								
emC_LUC[LUC_Num].SCADA.Out.OperatorMd	:=	emC_LUC[LUC_Num].SM.Out.OperatorMd		;
emC_LUC[LUC_Num].SCADA.Out.AutoMd	:=	emC_LUC[LUC_Num].SM.Out.AutoMd		;
emC_LUC[LUC_Num].SCADA.Out.ManualMd	:=	emC_LUC[LUC_Num].SM.Out.ManualMd		;
emC_LUC[LUC_Num].SCADA.Out.FailedToStartAl	:=	emC_LUC[LUC_Num].SM.Out.FailedToStartAl		;
emC_LUC[LUC_Num].SCADA.Out.FailedToStopAl	:=	emC_LUC[LUC_Num].SM.Out.FailedToStopAl		;
emC_LUC[LUC_Num].SCADA.Out.NonCriticalAl	:=	emC_LUC[LUC_Num].SM.In.NonCriticalAlarm		;
emC_LUC[LUC_Num].SCADA.Out.WarningAl	:=	emC_LUC[LUC_Num].SM.In.Warning		;
emC_LUC[LUC_Num].SCADA.Out.CriticalAl	:=	emC_LUC[LUC_Num].SM.In.CriticalAlarm		;
emC_LUC[LUC_Num].SCADA.Out.HealthySt	:=	emC_LUC[LUC_Num].SM.In.HealthySt		;
emC_LUC[LUC_Num].SCADA.Out.OnlineSt	:=	emC_LUC[LUC_Num].SM.In.OnlineSt		;
emC_LUC[LUC_Num].SCADA.Out.RunningSt	:=	emC_LUC[LUC_Num].SM.In.RunningSt		;
emC_LUC[LUC_Num].SCADA.Out.BatEmergencyStop	:=	emC_LUC[LUC_Num].BattPLC.CtrlLo.Out.Batt_Sys.Alarm.EStopAl     		;
emC_LUC[LUC_Num].SCADA.Out.BatInitializeSt	:=	emC_LUC[LUC_Num].BattPLC.CtrlLo.Out.Batt_Sys.BattSMState.BatInitializeSt		;
emC_LUC[LUC_Num].SCADA.Out.BatNotReadySt	:=	emC_LUC[LUC_Num].BattPLC.CtrlLo.Out.Batt_Sys.BattSMState.BatNotReadySt		;
emC_LUC[LUC_Num].SCADA.Out.BatReadySt	:=	emC_LUC[LUC_Num].BattPLC.CtrlLo.Out.Batt_Sys.BattSMState.BatReadySt		;
emC_LUC[LUC_Num].SCADA.Out.BatStartingSt	:=	emC_LUC[LUC_Num].BattPLC.CtrlLo.Out.Batt_Sys.BattSMState.BatStartingSt		;
emC_LUC[LUC_Num].SCADA.Out.BatOnlineSt	:=	emC_LUC[LUC_Num].BattPLC.CtrlLo.Out.Batt_Sys.BattSMState.BatOnlineSt		;
emC_LUC[LUC_Num].SCADA.Out.BatStoppingSt	:=	emC_LUC[LUC_Num].BattPLC.CtrlLo.Out.Batt_Sys.BattSMState.BatStoppingSt		;
emC_LUC[LUC_Num].SCADA.Out.BmsChargingSt	:=	emC_LUC[LUC_Num].BattPLC.CtrlLo.Out.Batt_Sys.BMS_Mode.ChargingSt     		;
emC_LUC[LUC_Num].SCADA.Out.BmsDischargingSt	:=	emC_LUC[LUC_Num].BattPLC.CtrlLo.Out.Batt_Sys.BMS_Mode.DischargingSt     		;
emC_LUC[LUC_Num].SCADA.Out.BattRunningSt	:=	emC_LUC[LUC_Num].BattPLC.CtrlLo.Out.Batt_Sys.BMS_Mode.BattRunningSt     		;
emC_LUC[LUC_Num].SCADA.Out.BmsRkPartOnlineSt	:=	emC_LUC[LUC_Num].BattPLC.CtrlLo.Out.Batt_Sys.BMS_Mode.RkPartOnlineSt     		;
emC_LUC[LUC_Num].SCADA.Out.BmsEStopSPDSt	:=	emC_LUC[LUC_Num].BattPLC.CtrlLo.Out.Batt_Sys.BMS_Mode.EStopSPDSt     		;
emC_LUC[LUC_Num].SCADA.Out.BmsEStopProtSt	:=	emC_LUC[LUC_Num].BattPLC.CtrlLo.Out.Batt_Sys.BMS_Mode.EStopProtSt     		;
emC_LUC[LUC_Num].SCADA.Out.BmsEStopPartSt	:=	emC_LUC[LUC_Num].BattPLC.CtrlLo.Out.Batt_Sys.BMS_Mode.EStopPartSt     		;
emC_LUC[LUC_Num].SCADA.Out.BmsHealthySt	:=	emC_LUC[LUC_Num].BattPLC.CtrlLo.Out.Batt_Sys.Alarm.HealthySt     		;
emC_LUC[LUC_Num].SCADA.Out.BmsFireSysOkSt	:=	emC_LUC[LUC_Num].BattPLC.CtrlLo.Out.Batt_Sys.Alarm.FireSysOkSt     		;
emC_LUC[LUC_Num].SCADA.Out.BmsCriticalAl	:=	emC_LUC[LUC_Num].BattPLC.CtrlLo.Out.Batt_Sys.Alarm.CriticalAl		;
emC_LUC[LUC_Num].SCADA.Out.BmsNonCriticalAl	:=	emC_LUC[LUC_Num].BattPLC.CtrlLo.Out.Batt_Sys.Alarm.NonCriticalAl		;
emC_LUC[LUC_Num].SCADA.Out.BmsWarningAl	:=	emC_LUC[LUC_Num].BattPLC.CtrlLo.Out.Batt_Sys.Alarm.WarningAl		;
emC_LUC[LUC_Num].SCADA.Out.BmsStateTOUT	:=	emC_LUC[LUC_Num].BattPLC.CtrlLo.Out.Batt_Sys.Alarm.StateTOUT		;
emC_LUC[LUC_Num].SCADA.Out.BmsInitCommsFail	:=	emC_LUC[LUC_Num].BattPLC.CtrlLo.Out.Batt_Sys.Alarm.InitCommsFail		;
emC_LUC[LUC_Num].SCADA.Out.BmsMinRkCloseFail	:=	emC_LUC[LUC_Num].BattPLC.CtrlLo.Out.Batt_Sys.Alarm.MinRkCloseFail		;
emC_LUC[LUC_Num].SCADA.Out.BmsRkTripStart	:=	emC_LUC[LUC_Num].BattPLC.CtrlLo.Out.Batt_Sys.Alarm.RkTripStart		;
emC_LUC[LUC_Num].SCADA.Out.BmsMinRkOnlineFail	:=	emC_LUC[LUC_Num].BattPLC.CtrlLo.Out.Batt_Sys.Alarm.MinRkOnlineFail		;
emC_LUC[LUC_Num].SCADA.Out.BmsRkFailToOpen	:=	emC_LUC[LUC_Num].BattPLC.CtrlLo.Out.Batt_Sys.Alarm.RkFailToOpen		;
emC_LUC[LUC_Num].SCADA.Out.BmsSysFireAl	:=	emC_LUC[LUC_Num].BattPLC.CtrlLo.Out.Batt_Sys.Alarm.SysFireAl		;
emC_LUC[LUC_Num].SCADA.Out.BmsBmsLostCommsAl	:=	emC_LUC[LUC_Num].BattPLC.CtrlLo.Out.Batt_Sys.Alarm.BmsLostCommsAl		;
emC_LUC[LUC_Num].SCADA.Out.BmsBankFault	:=	emC_LUC[LUC_Num].BattPLC.CtrlLo.Out.Batt_Sys.Alarm.BankFault		;
emC_LUC[LUC_Num].SCADA.Out.BmsEStopAl	:=	emC_LUC[LUC_Num].BattPLC.CtrlLo.Out.Batt_Sys.Alarm.EStopAl		;
emC_LUC[LUC_Num].SCADA.Out.BmsExtReadyStNotSetAl	:=	emC_LUC[LUC_Num].BattPLC.CtrlLo.Out.Batt_Sys.Alarm.ExtReadyStNotSetAl		;
emC_LUC[LUC_Num].SCADA.Out.BattUSyncErrAl	:=	emC_LUC[LUC_Num].BattPLC.CtrlLo.Out.Batt_Sys.Alarm.BattUSyncErrAl		;
emC_LUC[LUC_Num].SCADA.Out.BmsRkFail2Cls	:=	emC_LUC[LUC_Num].BattPLC.CtrlLo.Out.Batt_Sys.Alarm.RkFail2Cls		;
emC_LUC[LUC_Num].SCADA.Out.BmsRkCntrFailAl	:=	emC_LUC[LUC_Num].BattPLC.CtrlLo.Out.Batt_Sys.Alarm.RkCntrFailAl		;
emC_LUC[LUC_Num].SCADA.Out.BmsRTUComAl	:=	emC_LUC[LUC_Num].BattPLC.CtrlLo.Out.Batt_Sys.BMSAlarmSummary.RTUComAl		;
emC_LUC[LUC_Num].SCADA.Out.BmsRTUComFlt	:=	emC_LUC[LUC_Num].BattPLC.CtrlLo.Out.Batt_Sys.BMSAlarmSummary.RTUComFlt		;
emC_LUC[LUC_Num].SCADA.Out.BmsRkVoltImbAl	:=	emC_LUC[LUC_Num].BattPLC.CtrlLo.Out.Batt_Sys.BMSAlarmSummary.RkVoltImbAl		;
emC_LUC[LUC_Num].SCADA.Out.BmsSysStopAl	:=	emC_LUC[LUC_Num].BattPLC.CtrlLo.Out.Batt_Sys.BMSAlarmSummary.SysStopAl		;
emC_LUC[LUC_Num].SCADA.Out.BmsModuleUnderTempAl	:=	emC_LUC[LUC_Num].BattPLC.CtrlLo.Out.Batt_Sys.BMSAlarm.ModuleUnderTempAl		;
emC_LUC[LUC_Num].SCADA.Out.BmsModuleOverTempAl	:=	emC_LUC[LUC_Num].BattPLC.CtrlLo.Out.Batt_Sys.BMSAlarm.ModuleOverTempAl		;
emC_LUC[LUC_Num].SCADA.Out.BmsModuleUnVoltAl	:=	emC_LUC[LUC_Num].BattPLC.CtrlLo.Out.Batt_Sys.BMSAlarm.ModuleUnVoltAl		;
emC_LUC[LUC_Num].SCADA.Out.BmsModuleOvVoltAl	:=	emC_LUC[LUC_Num].BattPLC.CtrlLo.Out.Batt_Sys.BMSAlarm.ModuleOvVoltAl		;
emC_LUC[LUC_Num].SCADA.Out.BmsRackVoltRegAl	:=	emC_LUC[LUC_Num].BattPLC.CtrlLo.Out.Batt_Sys.BMSAlarm.RackVoltRegAl		;
emC_LUC[LUC_Num].SCADA.Out.BmsRackTempRegAl	:=	emC_LUC[LUC_Num].BattPLC.CtrlLo.Out.Batt_Sys.BMSAlarm.RackTempRegAl		;
emC_LUC[LUC_Num].SCADA.Out.BmsAuxProtAl	:=	emC_LUC[LUC_Num].BattPLC.CtrlLo.Out.Batt_Sys.BMSAlarm.AuxProtAl		;
emC_LUC[LUC_Num].SCADA.Out.BmsChargeOperLimAl	:=	emC_LUC[LUC_Num].BattPLC.CtrlLo.Out.Batt_Sys.BMSAlarm.ChargeOperLimAl		;
emC_LUC[LUC_Num].SCADA.Out.BmsDischargeOperLimAl	:=	emC_LUC[LUC_Num].BattPLC.CtrlLo.Out.Batt_Sys.BMSAlarm.DischargeOperLimAl		;
emC_LUC[LUC_Num].SCADA.Out.BmsRackUnVoltAl	:=	emC_LUC[LUC_Num].BattPLC.CtrlLo.Out.Batt_Sys.BMSAlarm.RackUnVoltAl		;
emC_LUC[LUC_Num].SCADA.Out.BmsRackOvVoltAl	:=	emC_LUC[LUC_Num].BattPLC.CtrlLo.Out.Batt_Sys.BMSAlarm.RackOvVoltAl		;
emC_LUC[LUC_Num].SCADA.Out.BmsRackCommsAl	:=	emC_LUC[LUC_Num].BattPLC.CtrlLo.Out.Batt_Sys.BMSAlarm.RackCommsAl		;
emC_LUC[LUC_Num].SCADA.Out.BmsTrayCommsAl	:=	emC_LUC[LUC_Num].BattPLC.CtrlLo.Out.Batt_Sys.BMSAlarm.TrayCommsAl		;
emC_LUC[LUC_Num].SCADA.Out.BmsDcCntrSensor1Al	:=	emC_LUC[LUC_Num].BattPLC.CtrlLo.Out.Batt_Sys.BMSAlarm.DcCntrSensor1Al		;
emC_LUC[LUC_Num].SCADA.Out.BmsDcCntrSensor2Al	:=	emC_LUC[LUC_Num].BattPLC.CtrlLo.Out.Batt_Sys.BMSAlarm.DcCntrSensor2Al		;
emC_LUC[LUC_Num].SCADA.Out.BmsFanFailAl	:=	emC_LUC[LUC_Num].BattPLC.CtrlLo.Out.Batt_Sys.BMSAlarm.FanFailAl		;
emC_LUC[LUC_Num].SCADA.Out.BmsChargeOverCurrentAl	:=	emC_LUC[LUC_Num].BattPLC.CtrlLo.Out.Batt_Sys.BMSAlarm.ChargeOverCurrentAl		;
emC_LUC[LUC_Num].SCADA.Out.BmsDisChargeOverCurrentAl	:=	emC_LUC[LUC_Num].BattPLC.CtrlLo.Out.Batt_Sys.BMSAlarm.DisChargeOverCurrentAl		;
emC_LUC[LUC_Num].SCADA.Out.BmsRackVSenseDiffAl	:=	emC_LUC[LUC_Num].BattPLC.CtrlLo.Out.Batt_Sys.BMSAlarm.RackVSenseDiffAl		;
emC_LUC[LUC_Num].SCADA.Out.BmsRackFuseFailAl	:=	emC_LUC[LUC_Num].BattPLC.CtrlLo.Out.Batt_Sys.BMSAlarm.RackFuseFailAl		;
emC_LUC[LUC_Num].SCADA.Out.BmsRackCurrentSenserFailAl	:=	emC_LUC[LUC_Num].BattPLC.CtrlLo.Out.Batt_Sys.BMSAlarm.RackCurrentSenserFailAl		;
emC_LUC[LUC_Num].SCADA.Out.BmsRackPermanentUVAl	:=	emC_LUC[LUC_Num].BattPLC.CtrlLo.Out.Batt_Sys.BMSAlarm.RackPermanentUVAl		;
emC_LUC[LUC_Num].SCADA.Out.BmsDcCntr1Al	:=	emC_LUC[LUC_Num].BattPLC.CtrlLo.Out.Batt_Sys.BMSAlarm.DcCntr1Al		;
emC_LUC[LUC_Num].SCADA.Out.BmsDcCntr2Al	:=	emC_LUC[LUC_Num].BattPLC.CtrlLo.Out.Batt_Sys.BMSAlarm.DcCntr2Al		;
emC_LUC[LUC_Num].SCADA.Out.BmsDcSwCntFailAl	:=	emC_LUC[LUC_Num].BattPLC.CtrlLo.Out.Batt_Sys.BMSAlarm.DcSwCntFailAl		;
emC_LUC[LUC_Num].SCADA.Out.BmsCellVoltSenFailAl	:=	emC_LUC[LUC_Num].BattPLC.CtrlLo.Out.Batt_Sys.BMSAlarm.CellVoltSenFailAl		;
emC_LUC[LUC_Num].SCADA.Out.BmsDCFuseSenserFailAl	:=	emC_LUC[LUC_Num].BattPLC.CtrlLo.Out.Batt_Sys.BMSAlarm.DCFuseSenserFailAl		;
emC_LUC[LUC_Num].SCADA.Out.BmsModuleUnderTempProt	:=	emC_LUC[LUC_Num].BattPLC.CtrlLo.Out.Batt_Sys.BMSProt.ModuleUnderTempAl		;
emC_LUC[LUC_Num].SCADA.Out.BmsModuleOverTempProt	:=	emC_LUC[LUC_Num].BattPLC.CtrlLo.Out.Batt_Sys.BMSProt.ModuleOverTempAl		;
emC_LUC[LUC_Num].SCADA.Out.BmsModuleUnVoltProt	:=	emC_LUC[LUC_Num].BattPLC.CtrlLo.Out.Batt_Sys.BMSProt.ModuleUnVoltAl		;
emC_LUC[LUC_Num].SCADA.Out.BmsModuleOvVoltProt	:=	emC_LUC[LUC_Num].BattPLC.CtrlLo.Out.Batt_Sys.BMSProt.ModuleOvVoltAl		;
emC_LUC[LUC_Num].SCADA.Out.BmsRackVoltRegProt	:=	emC_LUC[LUC_Num].BattPLC.CtrlLo.Out.Batt_Sys.BMSProt.RackVoltRegAl		;
emC_LUC[LUC_Num].SCADA.Out.BmsRackTempRegProt	:=	emC_LUC[LUC_Num].BattPLC.CtrlLo.Out.Batt_Sys.BMSProt.RackTempRegAl		;
emC_LUC[LUC_Num].SCADA.Out.BmsAuxProtProt	:=	emC_LUC[LUC_Num].BattPLC.CtrlLo.Out.Batt_Sys.BMSProt.AuxProtAl		;
emC_LUC[LUC_Num].SCADA.Out.BmsChargeOperLimProt	:=	emC_LUC[LUC_Num].BattPLC.CtrlLo.Out.Batt_Sys.BMSProt.ChargeOperLimAl		;
emC_LUC[LUC_Num].SCADA.Out.BmsDischargeOperLimProt	:=	emC_LUC[LUC_Num].BattPLC.CtrlLo.Out.Batt_Sys.BMSProt.DischargeOperLimAl		;
emC_LUC[LUC_Num].SCADA.Out.BmsRackUnVoltProt	:=	emC_LUC[LUC_Num].BattPLC.CtrlLo.Out.Batt_Sys.BMSProt.RackUnVoltAl		;
emC_LUC[LUC_Num].SCADA.Out.BmsRackOvVoltProt	:=	emC_LUC[LUC_Num].BattPLC.CtrlLo.Out.Batt_Sys.BMSProt.RackOvVoltAl		;
emC_LUC[LUC_Num].SCADA.Out.BmsRackCommsProt	:=	emC_LUC[LUC_Num].BattPLC.CtrlLo.Out.Batt_Sys.BMSProt.RackCommsAl		;
emC_LUC[LUC_Num].SCADA.Out.BmsTrayCommsProt	:=	emC_LUC[LUC_Num].BattPLC.CtrlLo.Out.Batt_Sys.BMSProt.TrayCommsAl		;
emC_LUC[LUC_Num].SCADA.Out.BmsDcCntrSensor1Prot	:=	emC_LUC[LUC_Num].BattPLC.CtrlLo.Out.Batt_Sys.BMSProt.DcCntrSensor1Al		;
emC_LUC[LUC_Num].SCADA.Out.BmsDcCntrSensor2Prot	:=	emC_LUC[LUC_Num].BattPLC.CtrlLo.Out.Batt_Sys.BMSProt.DcCntrSensor2Al		;
emC_LUC[LUC_Num].SCADA.Out.BmsFanFailProt	:=	emC_LUC[LUC_Num].BattPLC.CtrlLo.Out.Batt_Sys.BMSProt.FanFailAl		;
emC_LUC[LUC_Num].SCADA.Out.BmsChargeOverCurrentProt	:=	emC_LUC[LUC_Num].BattPLC.CtrlLo.Out.Batt_Sys.BMSProt.ChargeOverCurrentAl		;
emC_LUC[LUC_Num].SCADA.Out.BmsDisChargeOverCurrentProt	:=	emC_LUC[LUC_Num].BattPLC.CtrlLo.Out.Batt_Sys.BMSProt.DisChargeOverCurrentAl		;
emC_LUC[LUC_Num].SCADA.Out.BmsRackVSenseDiffProt	:=	emC_LUC[LUC_Num].BattPLC.CtrlLo.Out.Batt_Sys.BMSProt.RackVSenseDiffAl		;
emC_LUC[LUC_Num].SCADA.Out.BmsRackFuseFailProt	:=	emC_LUC[LUC_Num].BattPLC.CtrlLo.Out.Batt_Sys.BMSProt.RackFuseFailAl		;
emC_LUC[LUC_Num].SCADA.Out.BmsRackCurrentSenserFailProt	:=	emC_LUC[LUC_Num].BattPLC.CtrlLo.Out.Batt_Sys.BMSProt.RackCurrentSenserFailAl		;
emC_LUC[LUC_Num].SCADA.Out.BmsRackPermanentUVProt	:=	emC_LUC[LUC_Num].BattPLC.CtrlLo.Out.Batt_Sys.BMSProt.RackPermanentUVAl		;
emC_LUC[LUC_Num].SCADA.Out.BmsDcCntr1Prot	:=	emC_LUC[LUC_Num].BattPLC.CtrlLo.Out.Batt_Sys.BMSProt.DcCntr1Al		;
emC_LUC[LUC_Num].SCADA.Out.BmsDcCntr2Prot	:=	emC_LUC[LUC_Num].BattPLC.CtrlLo.Out.Batt_Sys.BMSProt.DcCntr2Al		;
emC_LUC[LUC_Num].SCADA.Out.BmsDcSwCntFailProt	:=	emC_LUC[LUC_Num].BattPLC.CtrlLo.Out.Batt_Sys.BMSProt.DcSwCntFailAl		;
emC_LUC[LUC_Num].SCADA.Out.BmsCellVoltSenFailProt	:=	emC_LUC[LUC_Num].BattPLC.CtrlLo.Out.Batt_Sys.BMSProt.CellVoltSenFailAl		;
emC_LUC[LUC_Num].SCADA.Out.BmsDCFuseSenserFailProt	:=	emC_LUC[LUC_Num].BattPLC.CtrlLo.Out.Batt_Sys.BMSProt.DCFuseSenserFailAl		;
								
for i:=1 to emC_LUC[LUC_Num].BattPLC.Pa.NbOfRackPa	DO	
	emC_LUC[LUC_Num].SCADA.Out.Rk[i].OnlineSt	:=	emC_LUC[LUC_Num].BattPLC.CtrlLo.Out.Batt_Rack.Batt_Rack_Array[i].Status.RkOnlineSt	;
	emC_LUC[LUC_Num].SCADA.Out.Rk[i].OnlineSt	:=	emC_LUC[LUC_Num].BattPLC.CtrlLo.Out.Batt_Rack.Batt_Rack_Array[i].Status.RkOnlineSt	;
	emC_LUC[LUC_Num].SCADA.Out.Rk[i].FaultSt	:=	emC_LUC[LUC_Num].BattPLC.CtrlLo.Out.Batt_Rack.Batt_Rack_Array[i].Alarm.RkCriticalAl OR emC_LUC[LUC_Num].BattPLC.CtrlLo.Out.Batt_Rack.Batt_Rack_Array[i].Alarm.RkNonCriticalAl ;
	emC_LUC[LUC_Num].SCADA.Out.Rk[i].SoCAct	:=	emC_LUC[LUC_Num].BattPLC.CtrlLo.Out.Batt_Rack.Batt_Rack_Array[i].Measure.SoCAct	;
	emC_LUC[LUC_Num].SCADA.Out.Rk[i].SoHAct	:=	emC_LUC[LUC_Num].BattPLC.CtrlLo.Out.Batt_Rack.Batt_Rack_Array[i].Measure.SoHAct	;
	emC_LUC[LUC_Num].SCADA.Out.Rk[i].UAct	:=	emC_LUC[LUC_Num].BattPLC.CtrlLo.Out.Batt_Rack.Batt_Rack_Array[i].Measure.UAct	;
	emC_LUC[LUC_Num].SCADA.Out.Rk[i].IAct	:=	emC_LUC[LUC_Num].BattPLC.CtrlLo.Out.Batt_Rack.Batt_Rack_Array[i].Measure.IAct	;
	emC_LUC[LUC_Num].SCADA.Out.Rk[i].TempAct	:=	emC_LUC[LUC_Num].BattPLC.CtrlLo.Out.Batt_Rack.Batt_Rack_Array[i].Measure.CellAvgTAct	;
END_FOR;
								
emC_LUC[LUC_Num].SCADA.Out.GCRunningSt	:=	emC_LUC[LUC_Num].emPs.PS.GCRunningSt		;
emC_LUC[LUC_Num].SCADA.Out.GCHealthy	:=	emC_LUC[LUC_Num].emPs.PS.GCHealthy		;
emC_LUC[LUC_Num].SCADA.Out.GCStartingSt	:=	emC_LUC[LUC_Num].emPs.PS.GCStartingSt		;
emC_LUC[LUC_Num].SCADA.Out.GCReadySt	:=	emC_LUC[LUC_Num].emPs.PS.GCReadySt		;
emC_LUC[LUC_Num].SCADA.Out.GCGridFollowing	:=	emC_LUC[LUC_Num].emPs.PS.GCGridFollowing		;
emC_LUC[LUC_Num].SCADA.Out.GCFaultSt	:=	emC_LUC[LUC_Num].emPs.PS.GCFaultSt		;
emC_LUC[LUC_Num].SCADA.Out.GCGridForming	:=	emC_LUC[LUC_Num].emPs.PS.GCGridForming		;
emC_LUC[LUC_Num].SCADA.Out.GCAreaEPSLost	:=	emC_LUC[LUC_Num].emPs.PS.GCAreaEPSLost		;
emC_LUC[LUC_Num].SCADA.Out.GCChargingSt	:=	emC_LUC[LUC_Num].emPs.PS.GCChargingSt		;
emC_LUC[LUC_Num].SCADA.Out.GCRideThru	:=	emC_LUC[LUC_Num].emPs.PS.GCRideThru		;
emC_LUC[LUC_Num].SCADA.Out.GCTransitionActiveSt	:=	emC_LUC[LUC_Num].emPs.PS.GCTransitionActiveSt		;
emC_LUC[LUC_Num].SCADA.Out.GCGndFault	:=	emC_LUC[LUC_Num].emPs.PS.GCGndFault		;
emC_LUC[LUC_Num].SCADA.Out.GCDCOverU	:=	emC_LUC[LUC_Num].emPs.PS.GCDCOverU		;
emC_LUC[LUC_Num].SCADA.Out.GCACDisconnect	:=	emC_LUC[LUC_Num].emPs.PS.GCACDisconnect		;
emC_LUC[LUC_Num].SCADA.Out.GCDCDisconnect	:=	emC_LUC[LUC_Num].emPs.PS.GCDCDisconnect		;
emC_LUC[LUC_Num].SCADA.Out.GCDCGridDisconnect	:=	emC_LUC[LUC_Num].emPs.PS.GCDCGridDisconnect		;
emC_LUC[LUC_Num].SCADA.Out.GCCabinetOpen	:=	emC_LUC[LUC_Num].emPs.PS.GCCabinetOpen		;
emC_LUC[LUC_Num].SCADA.Out.GCManualShutdown	:=	emC_LUC[LUC_Num].emPs.PS.GCManualShutdown		;
emC_LUC[LUC_Num].SCADA.Out.GCOverTemp	:=	emC_LUC[LUC_Num].emPs.PS.GCOverTemp		;
emC_LUC[LUC_Num].SCADA.Out.GCOverF	:=	emC_LUC[LUC_Num].emPs.PS.GCOverF		;
emC_LUC[LUC_Num].SCADA.Out.GCUnderF	:=	emC_LUC[LUC_Num].emPs.PS.GCUnderF		;
emC_LUC[LUC_Num].SCADA.Out.GCACOverVolt	:=	emC_LUC[LUC_Num].emPs.PS.GCACOverVolt		;
emC_LUC[LUC_Num].SCADA.Out.GCACUnderVolt	:=	emC_LUC[LUC_Num].emPs.PS.GCACUnderVolt		;
emC_LUC[LUC_Num].SCADA.Out.GCBlownFuse	:=	emC_LUC[LUC_Num].emPs.PS.GCBlownFuse		;
emC_LUC[LUC_Num].SCADA.Out.GCUnderTemp	:=	emC_LUC[LUC_Num].emPs.PS.GCUnderTemp		;
emC_LUC[LUC_Num].SCADA.Out.GCMemLoss	:=	emC_LUC[LUC_Num].emPs.PS.GCMemLoss		;
emC_LUC[LUC_Num].SCADA.Out.GCHWTestFailed	:=	emC_LUC[LUC_Num].emPs.PS.GCHWTestFailed		;
emC_LUC[LUC_Num].SCADA.Out.GCABBCtrlWrongConfig	:=	emC_LUC[LUC_Num].emPs.PS.GCABBCtrlWrongConfig		;
emC_LUC[LUC_Num].SCADA.Out.GCABBCtrlReady	:=	emC_LUC[LUC_Num].emPs.PS.GCABBCtrlReady		;
emC_LUC[LUC_Num].SCADA.Out.GCABBCtrlStartingSt	:=	emC_LUC[LUC_Num].emPs.PS.GCABBCtrlStartingSt		;
emC_LUC[LUC_Num].SCADA.Out.GCABBCtrlVGMActiveSt	:=	emC_LUC[LUC_Num].emPs.PS.GCABBCtrlVGMActiveSt		;
emC_LUC[LUC_Num].SCADA.Out.GCABBCtrlGSMActiveSt	:=	emC_LUC[LUC_Num].emPs.PS.GCABBCtrlGSMActiveSt		;
emC_LUC[LUC_Num].SCADA.Out.GCABBCtrlError	:=	emC_LUC[LUC_Num].emPs.PS.GCABBCtrlError		;
emC_LUC[LUC_Num].SCADA.Out.GCABBCtrlStoppingSt	:=	emC_LUC[LUC_Num].emPs.PS.GCABBCtrlStoppingSt		;
emC_LUC[LUC_Num].SCADA.Out.GCABBCtrlIslanded	:=	emC_LUC[LUC_Num].emPs.PS.GCABBCtrlIslanded		;
emC_LUC[LUC_Num].SCADA.Out.GCLostComms	:=	emC_LUC[LUC_Num].emPs.PS.GCLostComms		;
emC_LUC[LUC_Num].SCADA.Out.GCCommsOk	:=	emC_LUC[LUC_Num].emPs.PS.GCCommsOk		;
emC_LUC[LUC_Num].SCADA.Out.GCHardwareenablestatus	:=	emC_LUC[LUC_Num].emPs.PS.GCHardwareenablestatus		;
emC_LUC[LUC_Num].SCADA.Out.GCACPowerAvailable	:=	emC_LUC[LUC_Num].emPs.PS.GCACPowerAvailable		;
emC_LUC[LUC_Num].SCADA.Out.GCDCPowerAvailable	:=	emC_LUC[LUC_Num].emPs.PS.GCDCPowerAvailable		;
emC_LUC[LUC_Num].SCADA.Out.GCPowerCircuitEnabled	:=	emC_LUC[LUC_Num].emPs.PS.GCPowerCircuitEnabled		;
emC_LUC[LUC_Num].SCADA.Out.GCMX1relaystatus	:=	emC_LUC[LUC_Num].emPs.PS.GCMX1relaystatus		;
emC_LUC[LUC_Num].SCADA.Out.GCMX2relaystatus	:=	emC_LUC[LUC_Num].emPs.PS.GCMX2relaystatus		;
emC_LUC[LUC_Num].SCADA.Out.GCPrechargestatus	:=	emC_LUC[LUC_Num].emPs.PS.GCPrechargestatus		;
emC_LUC[LUC_Num].SCADA.Out.GCK2Relaystatus	:=	emC_LUC[LUC_Num].emPs.PS.GCK2Relaystatus		;
emC_LUC[LUC_Num].SCADA.Out.GCControlcommandsvalid	:=	emC_LUC[LUC_Num].emPs.PS.GCControlcommandsvalid		;
emC_LUC[LUC_Num].SCADA.Out.GCPowercommandValid	:=	emC_LUC[LUC_Num].emPs.PS.GCPowercommandValid		;
emC_LUC[LUC_Num].SCADA.Out.GCCurrentcommandValid	:=	emC_LUC[LUC_Num].emPs.PS.GCCurrentcommandValid		;
emC_LUC[LUC_Num].SCADA.Out.GCPhaserotationstatus	:=	emC_LUC[LUC_Num].emPs.PS.GCPhaserotationstatus		;
emC_LUC[LUC_Num].SCADA.Out.GCLinevoltagedetected	:=	emC_LUC[LUC_Num].emPs.PS.GCLinevoltagedetected		;
emC_LUC[LUC_Num].SCADA.Out.GCUnused	:=	emC_LUC[LUC_Num].emPs.PS.GCUnused		;
emC_LUC[LUC_Num].SCADA.Out.GCRemoteACPowerAvailable	:=	emC_LUC[LUC_Num].emPs.PS.GCRemoteACPowerAvailable		;
emC_LUC[LUC_Num].SCADA.Out.GCRemotephaserotationstatus	:=	emC_LUC[LUC_Num].emPs.PS.GCRemotephaserotationstatus		;
emC_LUC[LUC_Num].SCADA.Out.GCRemoteLineVoltageDetected	:=	emC_LUC[LUC_Num].emPs.PS.GCRemoteLineVoltageDetected		;
emC_LUC[LUC_Num].SCADA.Out.GCDI1Status	:=	emC_LUC[LUC_Num].emPs.PS.GCDI1Status		;
emC_LUC[LUC_Num].SCADA.Out.GCDI2Status	:=	emC_LUC[LUC_Num].emPs.PS.GCDI2Status		;
emC_LUC[LUC_Num].SCADA.Out.GCDI3Status	:=	emC_LUC[LUC_Num].emPs.PS.GCDI3Status		;
emC_LUC[LUC_Num].SCADA.Out.GCDI4Status	:=	emC_LUC[LUC_Num].emPs.PS.GCDI4Status		;
emC_LUC[LUC_Num].SCADA.Out.GCDO1Status	:=	emC_LUC[LUC_Num].emPs.PS.GCDO1Status		;
emC_LUC[LUC_Num].SCADA.Out.GCDO2Status	:=	emC_LUC[LUC_Num].emPs.PS.GCDO2Status		;
emC_LUC[LUC_Num].SCADA.Out.GCDO3Status	:=	emC_LUC[LUC_Num].emPs.PS.GCDO3Status		;
emC_LUC[LUC_Num].SCADA.Out.GCDO4Status	:=	emC_LUC[LUC_Num].emPs.PS.GCDO4Status		;
emC_LUC[LUC_Num].SCADA.Out.GCDClinkRefCmdValid	:=	emC_LUC[LUC_Num].emPs.PS.GCDClinkRefCmdValid		;
emC_LUC[LUC_Num].SCADA.Out.GCPumpRunning	:=	emC_LUC[LUC_Num].emPs.PS.GCPumpRunning		;
emC_LUC[LUC_Num].SCADA.Out.GCPumpFault	:=	emC_LUC[LUC_Num].emPs.PS.GCPumpFault		;
emC_LUC[LUC_Num].SCADA.Out.GCABBLostCommsStop	:=	emC_LUC[LUC_Num].emPs.PS.GCABBLostCommsStop		;
emC_LUC[LUC_Num].SCADA.Out.GCCtrlSystemReady	:=	emC_LUC[LUC_Num].emPs.PS.CtrlSystemReady		;
emC_LUC[LUC_Num].SCADA.Out.GCFlt_Estp	:=	emC_LUC[LUC_Num].emPs.PS.GCFltFlgs.Estp		;
emC_LUC[LUC_Num].SCADA.Out.GCFlt_ACOverCurrent	:=	emC_LUC[LUC_Num].emPs.PS.GCFltFlgs.ACOverCurrent		;
emC_LUC[LUC_Num].SCADA.Out.GCFlt_DCOverCurrent	:=	emC_LUC[LUC_Num].emPs.PS.GCFltFlgs.DCOverCurrent		;
emC_LUC[LUC_Num].SCADA.Out.GCFlt_DCOverVoltage	:=	emC_LUC[LUC_Num].emPs.PS.GCFltFlgs.DCOverVoltage		;
emC_LUC[LUC_Num].SCADA.Out.GCFlt_PDOverTemp	:=	emC_LUC[LUC_Num].emPs.PS.GCFltFlgs.PDOverTemp		;
emC_LUC[LUC_Num].SCADA.Out.GCFlt_InvOverTemp	:=	emC_LUC[LUC_Num].emPs.PS.GCFltFlgs.InvOverTemp		;
emC_LUC[LUC_Num].SCADA.Out.GCFlt_CmdMsg	:=	emC_LUC[LUC_Num].emPs.PS.GCFltFlgs.CmdMsg		;
emC_LUC[LUC_Num].SCADA.Out.GCFlt_DCUnderVolt	:=	emC_LUC[LUC_Num].emPs.PS.GCFltFlgs.DCUnderVolt		;
emC_LUC[LUC_Num].SCADA.Out.GCFlt_ACOverVolt	:=	emC_LUC[LUC_Num].emPs.PS.GCFltFlgs.ACOverVolt		;
emC_LUC[LUC_Num].SCADA.Out.GCFlt_IllegalTrans	:=	emC_LUC[LUC_Num].emPs.PS.GCFltFlgs.IllegalTrans		;
emC_LUC[LUC_Num].SCADA.Out.GCFlt_EEHeat	:=	emC_LUC[LUC_Num].emPs.PS.GCFltFlgs.EEHeat		;
emC_LUC[LUC_Num].SCADA.Out.GCFlt_EESction	:=	emC_LUC[LUC_Num].emPs.PS.GCFltFlgs.EESction		;
emC_LUC[LUC_Num].SCADA.Out.GCFlt_Cool	:=	emC_LUC[LUC_Num].emPs.PS.GCFltFlgs.Cool		;
emC_LUC[LUC_Num].SCADA.Out.GCFlt_TimedOverLoadAC	:=	emC_LUC[LUC_Num].emPs.PS.GCFltFlgs.TimedOverLoadAC		;
emC_LUC[LUC_Num].SCADA.Out.GCFlt_TimedOverLoadDC	:=	emC_LUC[LUC_Num].emPs.PS.GCFltFlgs.TimedOverLoadDC		;
emC_LUC[LUC_Num].SCADA.Out.GCFlt_ICOL	:=	emC_LUC[LUC_Num].emPs.PS.GCFltFlgs.ICOL		;
emC_LUC[LUC_Num].SCADA.Out.GCFlt_CtlBdVolt	:=	emC_LUC[LUC_Num].emPs.PS.GCFltFlgs.CtlBdVolt		;
emC_LUC[LUC_Num].SCADA.Out.GCFlt_PChImbal	:=	emC_LUC[LUC_Num].emPs.PS.GCFltFlgs.PChImbal		;
emC_LUC[LUC_Num].SCADA.Out.GCFlt_DiDt	:=	emC_LUC[LUC_Num].emPs.PS.GCFltFlgs.DiDt		;
emC_LUC[LUC_Num].SCADA.Out.GCFlt_CoolingFlw	:=	emC_LUC[LUC_Num].emPs.PS.GCFltFlgs.CoolingFlw		;
emC_LUC[LUC_Num].SCADA.Out.GCFlt_ThrmOverLoad	:=	emC_LUC[LUC_Num].emPs.PS.GCFltFlgs.ThrmOverLoad		;
emC_LUC[LUC_Num].SCADA.Out.GCFlt_Fan	:=	emC_LUC[LUC_Num].emPs.PS.GCFltFlgs.Fan		;
emC_LUC[LUC_Num].SCADA.Out.GCFlt_POR	:=	emC_LUC[LUC_Num].emPs.PS.GCFltFlgs.POR		;
emC_LUC[LUC_Num].SCADA.Out.GCFlt_Condensation	:=	emC_LUC[LUC_Num].emPs.PS.GCFltFlgs.Condensation		;
emC_LUC[LUC_Num].SCADA.Out.GCFlt_I2C	:=	emC_LUC[LUC_Num].emPs.PS.GCFltFlgs.I2C		;
emC_LUC[LUC_Num].SCADA.Out.GCFlt_ExternalInhibit	:=	emC_LUC[LUC_Num].emPs.PS.GCFltFlgs.ExternalInhibit		;
emC_LUC[LUC_Num].SCADA.Out.GCFlt_GroundFault	:=	emC_LUC[LUC_Num].emPs.PS.GCFltFlgs.GroundFault		;
emC_LUC[LUC_Num].SCADA.Out.GCFlt_Fuse	:=	emC_LUC[LUC_Num].emPs.PS.GCFltFlgs.Fuse		;
emC_LUC[LUC_Num].SCADA.Out.GCFlt_Rsvd28	:=	emC_LUC[LUC_Num].emPs.PS.GCFltFlgs.Rsvd28		;
emC_LUC[LUC_Num].SCADA.Out.GCFlt_ACDisconnect	:=	emC_LUC[LUC_Num].emPs.PS.GCFltFlgs.ACDisconnect		;
emC_LUC[LUC_Num].SCADA.Out.GCFlt_Rsvd30	:=	emC_LUC[LUC_Num].emPs.PS.GCFltFlgs.Rsvd30		;
emC_LUC[LUC_Num].SCADA.Out.GCFlt_Rsvd31	:=	emC_LUC[LUC_Num].emPs.PS.GCFltFlgs.Rsvd31		;
emC_LUC[LUC_Num].SCADA.Out.GCWrn_CANW	:=	emC_LUC[LUC_Num].emPs.PS.GCWrnFlgs.CANW		;
emC_LUC[LUC_Num].SCADA.Out.GCWrn_CANEP	:=	emC_LUC[LUC_Num].emPs.PS.GCWrnFlgs.CANEP		;
emC_LUC[LUC_Num].SCADA.Out.GCWrn_Thrm	:=	emC_LUC[LUC_Num].emPs.PS.GCWrnFlgs.Thrm		;
emC_LUC[LUC_Num].SCADA.Out.GCWrn_Fan	:=	emC_LUC[LUC_Num].emPs.PS.GCWrnFlgs.Fan		;
emC_LUC[LUC_Num].SCADA.Out.GCWrn_EeSaveActive	:=	emC_LUC[LUC_Num].emPs.PS.GCWrnFlgs.EeSaveActive		;
emC_LUC[LUC_Num].SCADA.Out.GCWrn_LocNetMismatch	:=	emC_LUC[LUC_Num].emPs.PS.GCWrnFlgs.LocNetMismatch		;
emC_LUC[LUC_Num].SCADA.Out.GCWrn_RemNetMismatch	:=	emC_LUC[LUC_Num].emPs.PS.GCWrnFlgs.RemNetMismatch		;
emC_LUC[LUC_Num].SCADA.Out.GCWrn_Condensation	:=	emC_LUC[LUC_Num].emPs.PS.GCWrnFlgs.Condensation		;
emC_LUC[LUC_Num].SCADA.Out.GCWrn_I2C	:=	emC_LUC[LUC_Num].emPs.PS.GCWrnFlgs.I2C		;
emC_LUC[LUC_Num].SCADA.Out.GCWrn_ExternalInhibit	:=	emC_LUC[LUC_Num].emPs.PS.GCWrnFlgs.ExternalInhibit		;
emC_LUC[LUC_Num].SCADA.Out.GCWrn_MaintReqd	:=	emC_LUC[LUC_Num].emPs.PS.GCWrnFlgs.MaintReqd		;
emC_LUC[LUC_Num].SCADA.Out.GCWrn_GroundFault	:=	emC_LUC[LUC_Num].emPs.PS.GCWrnFlgs.GroundFault		;
emC_LUC[LUC_Num].SCADA.Out.GCWrn_Fuse	:=	emC_LUC[LUC_Num].emPs.PS.GCWrnFlgs.Fuse		;
emC_LUC[LUC_Num].SCADA.Out.GCWrn_ACDisconnect	:=	emC_LUC[LUC_Num].emPs.PS.GCWrnFlgs.ACDisconnect		;
emC_LUC[LUC_Num].SCADA.Out.GCWrn_Rsvd14	:=	emC_LUC[LUC_Num].emPs.PS.GCWrnFlgs.Rsvd14		;
emC_LUC[LUC_Num].SCADA.Out.GCWrn_Rsvd15	:=	emC_LUC[LUC_Num].emPs.PS.GCWrnFlgs.Rsvd15		;
emC_LUC[LUC_Num].SCADA.Out.GCWrn_Rsvd16	:=	emC_LUC[LUC_Num].emPs.PS.GCWrnFlgs.Rsvd16		;
emC_LUC[LUC_Num].SCADA.Out.GCWrn_Rsvd17	:=	emC_LUC[LUC_Num].emPs.PS.GCWrnFlgs.Rsvd17		;
emC_LUC[LUC_Num].SCADA.Out.GCWrn_Rsvd18	:=	emC_LUC[LUC_Num].emPs.PS.GCWrnFlgs.Rsvd18		;
emC_LUC[LUC_Num].SCADA.Out.GCWrn_Rsvd19	:=	emC_LUC[LUC_Num].emPs.PS.GCWrnFlgs.Rsvd19		;
emC_LUC[LUC_Num].SCADA.Out.GCWrn_Rsvd20	:=	emC_LUC[LUC_Num].emPs.PS.GCWrnFlgs.Rsvd20		;
emC_LUC[LUC_Num].SCADA.Out.GCWrn_Rsvd21	:=	emC_LUC[LUC_Num].emPs.PS.GCWrnFlgs.Rsvd21		;
emC_LUC[LUC_Num].SCADA.Out.GCWrn_Rsvd22	:=	emC_LUC[LUC_Num].emPs.PS.GCWrnFlgs.Rsvd22		;
emC_LUC[LUC_Num].SCADA.Out.GCWrn_Rsvd23	:=	emC_LUC[LUC_Num].emPs.PS.GCWrnFlgs.Rsvd23		;
emC_LUC[LUC_Num].SCADA.Out.GCWrn_Rsvd24	:=	emC_LUC[LUC_Num].emPs.PS.GCWrnFlgs.Rsvd24		;
emC_LUC[LUC_Num].SCADA.Out.GCWrn_Rsvd25	:=	emC_LUC[LUC_Num].emPs.PS.GCWrnFlgs.Rsvd25		;
emC_LUC[LUC_Num].SCADA.Out.GCWrn_Rsvd26	:=	emC_LUC[LUC_Num].emPs.PS.GCWrnFlgs.Rsvd26		;
emC_LUC[LUC_Num].SCADA.Out.GCWrn_Rsvd27	:=	emC_LUC[LUC_Num].emPs.PS.GCWrnFlgs.Rsvd27		;
emC_LUC[LUC_Num].SCADA.Out.GCWrn_Rsvd28	:=	emC_LUC[LUC_Num].emPs.PS.GCWrnFlgs.Rsvd28		;
emC_LUC[LUC_Num].SCADA.Out.GCWrn_Rsvd29	:=	emC_LUC[LUC_Num].emPs.PS.GCWrnFlgs.Rsvd29		;
emC_LUC[LUC_Num].SCADA.Out.GCWrn_Rsvd30	:=	emC_LUC[LUC_Num].emPs.PS.GCWrnFlgs.Rsvd30		;
emC_LUC[LUC_Num].SCADA.Out.GCCriticalAlarm	:=	emC_LUC[LUC_Num].emPs.PS.CriticalAlarm		;
emC_LUC[LUC_Num].SCADA.Out.GCNonCriticalAlarm	:=	emC_LUC[LUC_Num].emPs.PS.NonCriticalAlarm		;
emC_LUC[LUC_Num].SCADA.Out.GCWarning	:=	emC_LUC[LUC_Num].emPs.PS.Warning		;
emC_LUC[LUC_Num].SCADA.Out.GCreconnectDelay	:=	emC_LUC[LUC_Num].emPs.PS.GCreconnectDelay		;
emC_LUC[LUC_Num].SCADA.Out.GCMomentCessation	:=	emC_LUC[LUC_Num].emPs.PS.GCMomentCessation		;
emC_LUC[LUC_Num].SCADA.Out.GCInhibited	:=	emC_LUC[LUC_Num].emPs.PS.GCInhibited		;
								
								
								
								
								
								
S_SPI_MNG_1	(Digital_Feedback_Value:=	emC_LUC[LUC_Num].SCADA.Out.OperatorMd	,TimeTag:=Timestamp,IV:=FALSE);	OperatorMd_Q	:=	S_SPI_MNG_1.Digital_Feedback_Q	;
S_SPI_MNG_2	(Digital_Feedback_Value:=	emC_LUC[LUC_Num].SCADA.Out.AutoMd	,TimeTag:=Timestamp,IV:=FALSE);	AutoMd_Q	:=	S_SPI_MNG_2.Digital_Feedback_Q	;
S_SPI_MNG_3	(Digital_Feedback_Value:=	emC_LUC[LUC_Num].SCADA.Out.LocalOnlineSt	,TimeTag:=Timestamp,IV:=FALSE);	LocalOnlineSt_Q	:=	S_SPI_MNG_3.Digital_Feedback_Q	;
S_SPI_MNG_5	(Digital_Feedback_Value:=	emC_LUC[LUC_Num].SCADA.Out.ManualMd	,TimeTag:=Timestamp,IV:=FALSE);	ManualMd_Q	:=	S_SPI_MNG_5.Digital_Feedback_Q	;
S_SPI_MNG_6	(Digital_Feedback_Value:=	emC_LUC[LUC_Num].SCADA.Out.FailedToStartAl	,TimeTag:=Timestamp,IV:=FALSE);	FailedToStartAl_Q	:=	S_SPI_MNG_6.Digital_Feedback_Q	;
S_SPI_MNG_7	(Digital_Feedback_Value:=	emC_LUC[LUC_Num].SCADA.Out.FailedToStopAl	,TimeTag:=Timestamp,IV:=FALSE);	FailedToStopAl_Q	:=	S_SPI_MNG_7.Digital_Feedback_Q	;
S_SPI_MNG_8	(Digital_Feedback_Value:=	emC_LUC[LUC_Num].SCADA.Out.NonCriticalAl	,TimeTag:=Timestamp,IV:=FALSE);	NonCriticalAl_Q	:=	S_SPI_MNG_8.Digital_Feedback_Q	;
S_SPI_MNG_9	(Digital_Feedback_Value:=	emC_LUC[LUC_Num].SCADA.Out.WarningAl	,TimeTag:=Timestamp,IV:=FALSE);	WarningAl_Q	:=	S_SPI_MNG_9.Digital_Feedback_Q	;
S_SPI_MNG_10	(Digital_Feedback_Value:=	emC_LUC[LUC_Num].SCADA.Out.CriticalAl	,TimeTag:=Timestamp,IV:=FALSE);	CriticalAl_Q	:=	S_SPI_MNG_10.Digital_Feedback_Q	;
S_SPI_MNG_14	(Digital_Feedback_Value:=	emC_LUC[LUC_Num].SCADA.Out.EstopAl	,TimeTag:=Timestamp,IV:=FALSE);	EstopAl_Q	:=	S_SPI_MNG_14.Digital_Feedback_Q	;
S_SPI_MNG_19	(Digital_Feedback_Value:=	emC_LUC[LUC_Num].SCADA.Out.FaultAl	,TimeTag:=Timestamp,IV:=FALSE);	FaultAl_Q	:=	S_SPI_MNG_19.Digital_Feedback_Q	;
S_SPI_MNG_20	(Digital_Feedback_Value:=	emC_LUC[LUC_Num].SCADA.Out.HealthySt	,TimeTag:=Timestamp,IV:=FALSE);	HealthySt_Q	:=	S_SPI_MNG_20.Digital_Feedback_Q	;
S_SPI_MNG_21	(Digital_Feedback_Value:=	emC_LUC[LUC_Num].SCADA.Out.OnlineSt	,TimeTag:=Timestamp,IV:=FALSE);	OnlineSt_Q	:=	S_SPI_MNG_21.Digital_Feedback_Q	;
S_SPI_MNG_22	(Digital_Feedback_Value:=	emC_LUC[LUC_Num].SCADA.Out.RunningSt	,TimeTag:=Timestamp,IV:=FALSE);	RunningSt_Q	:=	S_SPI_MNG_22.Digital_Feedback_Q	;
S_SPI_MNG_23	(Digital_Feedback_Value:=	emC_LUC[LUC_Num].SCADA.Out.BatEmergencyStop	,TimeTag:=Timestamp,IV:=FALSE);	BatEmergencyStop_Q	:=	S_SPI_MNG_23.Digital_Feedback_Q	;
S_SPI_MNG_24	(Digital_Feedback_Value:=	emC_LUC[LUC_Num].SCADA.Out.BlackOutCondition	,TimeTag:=Timestamp,IV:=FALSE);	BlackOutCondition_Q	:=	S_SPI_MNG_24.Digital_Feedback_Q	;
S_SPI_MNG_25	(Digital_Feedback_Value:=	emC_LUC[LUC_Num].SCADA.Out.BatInitializeSt	,TimeTag:=Timestamp,IV:=FALSE);	BatInitializeSt_Q	:=	S_SPI_MNG_25.Digital_Feedback_Q	;
S_SPI_MNG_26	(Digital_Feedback_Value:=	emC_LUC[LUC_Num].SCADA.Out.BatNotReadySt	,TimeTag:=Timestamp,IV:=FALSE);	BatNotReadySt_Q	:=	S_SPI_MNG_26.Digital_Feedback_Q	;
S_SPI_MNG_27	(Digital_Feedback_Value:=	emC_LUC[LUC_Num].SCADA.Out.BatReadySt	,TimeTag:=Timestamp,IV:=FALSE);	BatReadySt_Q	:=	S_SPI_MNG_27.Digital_Feedback_Q	;
S_SPI_MNG_28	(Digital_Feedback_Value:=	emC_LUC[LUC_Num].SCADA.Out.BatStartingSt	,TimeTag:=Timestamp,IV:=FALSE);	BatStartingSt_Q	:=	S_SPI_MNG_28.Digital_Feedback_Q	;
S_SPI_MNG_29	(Digital_Feedback_Value:=	emC_LUC[LUC_Num].SCADA.Out.BatOnlineSt	,TimeTag:=Timestamp,IV:=FALSE);	BatOnlineSt_Q	:=	S_SPI_MNG_29.Digital_Feedback_Q	;
S_SPI_MNG_30	(Digital_Feedback_Value:=	emC_LUC[LUC_Num].SCADA.Out.BatStoppingSt	,TimeTag:=Timestamp,IV:=FALSE);	BatStoppingSt_Q	:=	S_SPI_MNG_30.Digital_Feedback_Q	;
S_SPI_MNG_31	(Digital_Feedback_Value:=	emC_LUC[LUC_Num].SCADA.Out.BmsEStopProtEn	,TimeTag:=Timestamp,IV:=FALSE);	BmsEStopProtEn_Q	:=	S_SPI_MNG_31.Digital_Feedback_Q	;
S_SPI_MNG_32	(Digital_Feedback_Value:=	emC_LUC[LUC_Num].SCADA.Out.BmsEStopSPDEn	,TimeTag:=Timestamp,IV:=FALSE);	BmsEStopSPDEn_Q	:=	S_SPI_MNG_32.Digital_Feedback_Q	;
S_SPI_MNG_33	(Digital_Feedback_Value:=	emC_LUC[LUC_Num].SCADA.Out.BmsChargingSt	,TimeTag:=Timestamp,IV:=FALSE);	BmsChargingSt_Q	:=	S_SPI_MNG_33.Digital_Feedback_Q	;
S_SPI_MNG_34	(Digital_Feedback_Value:=	emC_LUC[LUC_Num].SCADA.Out.BmsDischargingSt	,TimeTag:=Timestamp,IV:=FALSE);	BmsDischargingSt_Q	:=	S_SPI_MNG_34.Digital_Feedback_Q	;
S_SPI_MNG_35	(Digital_Feedback_Value:=	emC_LUC[LUC_Num].SCADA.Out.BattRunningSt	,TimeTag:=Timestamp,IV:=FALSE);	BattRunningSt_Q	:=	S_SPI_MNG_35.Digital_Feedback_Q	;
S_SPI_MNG_36	(Digital_Feedback_Value:=	emC_LUC[LUC_Num].SCADA.Out.BmsRkPartOnlineSt	,TimeTag:=Timestamp,IV:=FALSE);	BmsRkPartOnlineSt_Q	:=	S_SPI_MNG_36.Digital_Feedback_Q	;
S_SPI_MNG_37	(Digital_Feedback_Value:=	emC_LUC[LUC_Num].SCADA.Out.BmsEStopSPDSt	,TimeTag:=Timestamp,IV:=FALSE);	BmsEStopSPDSt_Q	:=	S_SPI_MNG_37.Digital_Feedback_Q	;
S_SPI_MNG_38	(Digital_Feedback_Value:=	emC_LUC[LUC_Num].SCADA.Out.BmsEStopProtSt	,TimeTag:=Timestamp,IV:=FALSE);	BmsEStopProtSt_Q	:=	S_SPI_MNG_38.Digital_Feedback_Q	;
S_SPI_MNG_39	(Digital_Feedback_Value:=	emC_LUC[LUC_Num].SCADA.Out.BmsEStopPartSt	,TimeTag:=Timestamp,IV:=FALSE);	BmsEStopPartSt_Q	:=	S_SPI_MNG_39.Digital_Feedback_Q	;
S_SPI_MNG_40	(Digital_Feedback_Value:=	emC_LUC[LUC_Num].SCADA.Out.BmsHealthySt	,TimeTag:=Timestamp,IV:=FALSE);	BmsHealthySt_Q	:=	S_SPI_MNG_40.Digital_Feedback_Q	;
S_SPI_MNG_41	(Digital_Feedback_Value:=	emC_LUC[LUC_Num].SCADA.Out.BmsFireSysOkSt	,TimeTag:=Timestamp,IV:=FALSE);	BmsFireSysOkSt_Q	:=	S_SPI_MNG_41.Digital_Feedback_Q	;
S_SPI_MNG_42	(Digital_Feedback_Value:=	emC_LUC[LUC_Num].SCADA.Out.BmsCriticalAl	,TimeTag:=Timestamp,IV:=FALSE);	BmsCriticalAl_Q	:=	S_SPI_MNG_42.Digital_Feedback_Q	;
S_SPI_MNG_43	(Digital_Feedback_Value:=	emC_LUC[LUC_Num].SCADA.Out.BmsNonCriticalAl	,TimeTag:=Timestamp,IV:=FALSE);	BmsNonCriticalAl_Q	:=	S_SPI_MNG_43.Digital_Feedback_Q	;
S_SPI_MNG_44	(Digital_Feedback_Value:=	emC_LUC[LUC_Num].SCADA.Out.BmsWarningAl	,TimeTag:=Timestamp,IV:=FALSE);	BmsWarningAl_Q	:=	S_SPI_MNG_44.Digital_Feedback_Q	;
S_SPI_MNG_45	(Digital_Feedback_Value:=	emC_LUC[LUC_Num].SCADA.Out.BmsStateTOUT	,TimeTag:=Timestamp,IV:=FALSE);	BmsStateTOUT_Q	:=	S_SPI_MNG_45.Digital_Feedback_Q	;
S_SPI_MNG_46	(Digital_Feedback_Value:=	emC_LUC[LUC_Num].SCADA.Out.BmsInitCommsFail	,TimeTag:=Timestamp,IV:=FALSE);	BmsInitCommsFail_Q	:=	S_SPI_MNG_46.Digital_Feedback_Q	;
S_SPI_MNG_47	(Digital_Feedback_Value:=	emC_LUC[LUC_Num].SCADA.Out.BmsMinRkCloseFail	,TimeTag:=Timestamp,IV:=FALSE);	BmsMinRkCloseFail_Q	:=	S_SPI_MNG_47.Digital_Feedback_Q	;
S_SPI_MNG_48	(Digital_Feedback_Value:=	emC_LUC[LUC_Num].SCADA.Out.BmsRkTripStart	,TimeTag:=Timestamp,IV:=FALSE);	BmsRkTripStart_Q	:=	S_SPI_MNG_48.Digital_Feedback_Q	;
S_SPI_MNG_49	(Digital_Feedback_Value:=	emC_LUC[LUC_Num].SCADA.Out.BmsMinRkOnlineFail	,TimeTag:=Timestamp,IV:=FALSE);	BmsMinRkOnlineFail_Q	:=	S_SPI_MNG_49.Digital_Feedback_Q	;
S_SPI_MNG_50	(Digital_Feedback_Value:=	emC_LUC[LUC_Num].SCADA.Out.BmsRkFailToOpen	,TimeTag:=Timestamp,IV:=FALSE);	BmsRkFailToOpen_Q	:=	S_SPI_MNG_50.Digital_Feedback_Q	;
S_SPI_MNG_51	(Digital_Feedback_Value:=	emC_LUC[LUC_Num].SCADA.Out.BmsSysFireAl	,TimeTag:=Timestamp,IV:=FALSE);	BmsSysFireAl_Q	:=	S_SPI_MNG_51.Digital_Feedback_Q	;
S_SPI_MNG_52	(Digital_Feedback_Value:=	emC_LUC[LUC_Num].SCADA.Out.BmsBmsLostCommsAl	,TimeTag:=Timestamp,IV:=FALSE);	BmsBmsLostCommsAl_Q	:=	S_SPI_MNG_52.Digital_Feedback_Q	;
S_SPI_MNG_53	(Digital_Feedback_Value:=	emC_LUC[LUC_Num].SCADA.Out.BmsBankFault	,TimeTag:=Timestamp,IV:=FALSE);	BmsBankFault_Q	:=	S_SPI_MNG_53.Digital_Feedback_Q	;
S_SPI_MNG_54	(Digital_Feedback_Value:=	emC_LUC[LUC_Num].SCADA.Out.BmsEStopAl	,TimeTag:=Timestamp,IV:=FALSE);	BmsEStopAl_Q	:=	S_SPI_MNG_54.Digital_Feedback_Q	;
S_SPI_MNG_55	(Digital_Feedback_Value:=	emC_LUC[LUC_Num].SCADA.Out.BmsExtReadyStNotSetAl	,TimeTag:=Timestamp,IV:=FALSE);	BmsExtReadyStNotSetAl_Q	:=	S_SPI_MNG_55.Digital_Feedback_Q	;
S_SPI_MNG_56	(Digital_Feedback_Value:=	emC_LUC[LUC_Num].SCADA.Out.BattUSyncErrAl	,TimeTag:=Timestamp,IV:=FALSE);	BattUSyncErrAl_Q	:=	S_SPI_MNG_56.Digital_Feedback_Q	;
S_SPI_MNG_57	(Digital_Feedback_Value:=	emC_LUC[LUC_Num].SCADA.Out.BmsRkFail2Cls	,TimeTag:=Timestamp,IV:=FALSE);	BmsRkFail2Cls_Q	:=	S_SPI_MNG_57.Digital_Feedback_Q	;
S_SPI_MNG_58	(Digital_Feedback_Value:=	emC_LUC[LUC_Num].SCADA.Out.BmsRkCntrFailAl	,TimeTag:=Timestamp,IV:=FALSE);	BmsRkCntrFailAl_Q	:=	S_SPI_MNG_58.Digital_Feedback_Q	;
S_SPI_MNG_59	(Digital_Feedback_Value:=	emC_LUC[LUC_Num].SCADA.Out.BmsRTUComAl	,TimeTag:=Timestamp,IV:=FALSE);	BmsRTUComAl_Q	:=	S_SPI_MNG_59.Digital_Feedback_Q	;
S_SPI_MNG_60	(Digital_Feedback_Value:=	emC_LUC[LUC_Num].SCADA.Out.BmsRTUComFlt	,TimeTag:=Timestamp,IV:=FALSE);	BmsRTUComFlt_Q	:=	S_SPI_MNG_60.Digital_Feedback_Q	;
S_SPI_MNG_61	(Digital_Feedback_Value:=	emC_LUC[LUC_Num].SCADA.Out.BmsRkVoltImbAl	,TimeTag:=Timestamp,IV:=FALSE);	BmsRkVoltImbAl_Q	:=	S_SPI_MNG_61.Digital_Feedback_Q	;
S_SPI_MNG_62	(Digital_Feedback_Value:=	emC_LUC[LUC_Num].SCADA.Out.BmsSysStopAl	,TimeTag:=Timestamp,IV:=FALSE);	BmsSysStopAl_Q	:=	S_SPI_MNG_62.Digital_Feedback_Q	;
S_SPI_MNG_63	(Digital_Feedback_Value:=	emC_LUC[LUC_Num].SCADA.Out.BmsModuleUnderTempAl	,TimeTag:=Timestamp,IV:=FALSE);	BmsModuleUnderTempAl_Q	:=	S_SPI_MNG_63.Digital_Feedback_Q	;
S_SPI_MNG_64	(Digital_Feedback_Value:=	emC_LUC[LUC_Num].SCADA.Out.BmsModuleOverTempAl	,TimeTag:=Timestamp,IV:=FALSE);	BmsModuleOverTempAl_Q	:=	S_SPI_MNG_64.Digital_Feedback_Q	;
S_SPI_MNG_65	(Digital_Feedback_Value:=	emC_LUC[LUC_Num].SCADA.Out.BmsModuleUnVoltAl	,TimeTag:=Timestamp,IV:=FALSE);	BmsModuleUnVoltAl_Q	:=	S_SPI_MNG_65.Digital_Feedback_Q	;
S_SPI_MNG_66	(Digital_Feedback_Value:=	emC_LUC[LUC_Num].SCADA.Out.BmsModuleOvVoltAl	,TimeTag:=Timestamp,IV:=FALSE);	BmsModuleOvVoltAl_Q	:=	S_SPI_MNG_66.Digital_Feedback_Q	;
S_SPI_MNG_67	(Digital_Feedback_Value:=	emC_LUC[LUC_Num].SCADA.Out.BmsRackVoltRegAl	,TimeTag:=Timestamp,IV:=FALSE);	BmsRackVoltRegAl_Q	:=	S_SPI_MNG_67.Digital_Feedback_Q	;
S_SPI_MNG_68	(Digital_Feedback_Value:=	emC_LUC[LUC_Num].SCADA.Out.BmsRackTempRegAl	,TimeTag:=Timestamp,IV:=FALSE);	BmsRackTempRegAl_Q	:=	S_SPI_MNG_68.Digital_Feedback_Q	;
S_SPI_MNG_69	(Digital_Feedback_Value:=	emC_LUC[LUC_Num].SCADA.Out.BmsAuxProtAl	,TimeTag:=Timestamp,IV:=FALSE);	BmsAuxProtAl_Q	:=	S_SPI_MNG_69.Digital_Feedback_Q	;
S_SPI_MNG_70	(Digital_Feedback_Value:=	emC_LUC[LUC_Num].SCADA.Out.BmsChargeOperLimAl	,TimeTag:=Timestamp,IV:=FALSE);	BmsChargeOperLimAl_Q	:=	S_SPI_MNG_70.Digital_Feedback_Q	;
S_SPI_MNG_71	(Digital_Feedback_Value:=	emC_LUC[LUC_Num].SCADA.Out.BmsDischargeOperLimAl	,TimeTag:=Timestamp,IV:=FALSE);	BmsDischargeOperLimAl_Q	:=	S_SPI_MNG_71.Digital_Feedback_Q	;
S_SPI_MNG_72	(Digital_Feedback_Value:=	emC_LUC[LUC_Num].SCADA.Out.BmsRackUnVoltAl	,TimeTag:=Timestamp,IV:=FALSE);	BmsRackUnVoltAl_Q	:=	S_SPI_MNG_72.Digital_Feedback_Q	;
S_SPI_MNG_73	(Digital_Feedback_Value:=	emC_LUC[LUC_Num].SCADA.Out.BmsRackOvVoltAl	,TimeTag:=Timestamp,IV:=FALSE);	BmsRackOvVoltAl_Q	:=	S_SPI_MNG_73.Digital_Feedback_Q	;
S_SPI_MNG_74	(Digital_Feedback_Value:=	emC_LUC[LUC_Num].SCADA.Out.BmsRackCommsAl	,TimeTag:=Timestamp,IV:=FALSE);	BmsRackCommsAl_Q	:=	S_SPI_MNG_74.Digital_Feedback_Q	;
S_SPI_MNG_75	(Digital_Feedback_Value:=	emC_LUC[LUC_Num].SCADA.Out.BmsTrayCommsAl	,TimeTag:=Timestamp,IV:=FALSE);	BmsTrayCommsAl_Q	:=	S_SPI_MNG_75.Digital_Feedback_Q	;
S_SPI_MNG_76	(Digital_Feedback_Value:=	emC_LUC[LUC_Num].SCADA.Out.BmsDcCntrSensor1Al	,TimeTag:=Timestamp,IV:=FALSE);	BmsDcCntrSensor1Al_Q	:=	S_SPI_MNG_76.Digital_Feedback_Q	;
S_SPI_MNG_77	(Digital_Feedback_Value:=	emC_LUC[LUC_Num].SCADA.Out.BmsDcCntrSensor2Al	,TimeTag:=Timestamp,IV:=FALSE);	BmsDcCntrSensor2Al_Q	:=	S_SPI_MNG_77.Digital_Feedback_Q	;
S_SPI_MNG_78	(Digital_Feedback_Value:=	emC_LUC[LUC_Num].SCADA.Out.BmsFanFailAl	,TimeTag:=Timestamp,IV:=FALSE);	BmsFanFailAl_Q	:=	S_SPI_MNG_78.Digital_Feedback_Q	;
S_SPI_MNG_79	(Digital_Feedback_Value:=	emC_LUC[LUC_Num].SCADA.Out.BmsChargeOverCurrentAl	,TimeTag:=Timestamp,IV:=FALSE);	BmsChargeOverCurrentAl_Q	:=	S_SPI_MNG_79.Digital_Feedback_Q	;
S_SPI_MNG_80	(Digital_Feedback_Value:=	emC_LUC[LUC_Num].SCADA.Out.BmsDisChargeOverCurrentAl	,TimeTag:=Timestamp,IV:=FALSE);	BmsDisChargeOverCurrentAl_Q	:=	S_SPI_MNG_80.Digital_Feedback_Q	;
S_SPI_MNG_81	(Digital_Feedback_Value:=	emC_LUC[LUC_Num].SCADA.Out.BmsRackVSenseDiffAl	,TimeTag:=Timestamp,IV:=FALSE);	BmsRackVSenseDiffAl_Q	:=	S_SPI_MNG_81.Digital_Feedback_Q	;
S_SPI_MNG_82	(Digital_Feedback_Value:=	emC_LUC[LUC_Num].SCADA.Out.BmsRackFuseFailAl	,TimeTag:=Timestamp,IV:=FALSE);	BmsRackFuseFailAl_Q	:=	S_SPI_MNG_82.Digital_Feedback_Q	;
S_SPI_MNG_83	(Digital_Feedback_Value:=	emC_LUC[LUC_Num].SCADA.Out.BmsRackCurrentSenserFailAl	,TimeTag:=Timestamp,IV:=FALSE);	BmsRackCurrentSenserFailAl_Q	:=	S_SPI_MNG_83.Digital_Feedback_Q	;
S_SPI_MNG_84	(Digital_Feedback_Value:=	emC_LUC[LUC_Num].SCADA.Out.BmsRackPermanentUVAl	,TimeTag:=Timestamp,IV:=FALSE);	BmsRackPermanentUVAl_Q	:=	S_SPI_MNG_84.Digital_Feedback_Q	;
S_SPI_MNG_85	(Digital_Feedback_Value:=	emC_LUC[LUC_Num].SCADA.Out.BmsDcCntr1Al	,TimeTag:=Timestamp,IV:=FALSE);	BmsDcCntr1Al_Q	:=	S_SPI_MNG_85.Digital_Feedback_Q	;
S_SPI_MNG_86	(Digital_Feedback_Value:=	emC_LUC[LUC_Num].SCADA.Out.BmsDcCntr2Al	,TimeTag:=Timestamp,IV:=FALSE);	BmsDcCntr2Al_Q	:=	S_SPI_MNG_86.Digital_Feedback_Q	;
S_SPI_MNG_87	(Digital_Feedback_Value:=	emC_LUC[LUC_Num].SCADA.Out.BmsDcSwCntFailAl	,TimeTag:=Timestamp,IV:=FALSE);	BmsDcSwCntFailAl_Q	:=	S_SPI_MNG_87.Digital_Feedback_Q	;
S_SPI_MNG_88	(Digital_Feedback_Value:=	emC_LUC[LUC_Num].SCADA.Out.BmsCellVoltSenFailAl	,TimeTag:=Timestamp,IV:=FALSE);	BmsCellVoltSenFailAl_Q	:=	S_SPI_MNG_88.Digital_Feedback_Q	;
S_SPI_MNG_89	(Digital_Feedback_Value:=	emC_LUC[LUC_Num].SCADA.Out.BmsDCFuseSenserFailAl	,TimeTag:=Timestamp,IV:=FALSE);	BmsDCFuseSenserFailAl_Q	:=	S_SPI_MNG_89.Digital_Feedback_Q	;
S_SPI_MNG_90	(Digital_Feedback_Value:=	emC_LUC[LUC_Num].SCADA.Out.BmsModuleUnderTempProt	,TimeTag:=Timestamp,IV:=FALSE);	BmsModuleUnderTempProt_Q	:=	S_SPI_MNG_90.Digital_Feedback_Q	;
S_SPI_MNG_91	(Digital_Feedback_Value:=	emC_LUC[LUC_Num].SCADA.Out.BmsModuleOverTempProt	,TimeTag:=Timestamp,IV:=FALSE);	BmsModuleOverTempProt_Q	:=	S_SPI_MNG_91.Digital_Feedback_Q	;
S_SPI_MNG_92	(Digital_Feedback_Value:=	emC_LUC[LUC_Num].SCADA.Out.BmsModuleUnVoltProt	,TimeTag:=Timestamp,IV:=FALSE);	BmsModuleUnVoltProt_Q	:=	S_SPI_MNG_92.Digital_Feedback_Q	;
S_SPI_MNG_93	(Digital_Feedback_Value:=	emC_LUC[LUC_Num].SCADA.Out.BmsModuleOvVoltProt	,TimeTag:=Timestamp,IV:=FALSE);	BmsModuleOvVoltProt_Q	:=	S_SPI_MNG_93.Digital_Feedback_Q	;
S_SPI_MNG_94	(Digital_Feedback_Value:=	emC_LUC[LUC_Num].SCADA.Out.BmsRackVoltRegProt	,TimeTag:=Timestamp,IV:=FALSE);	BmsRackVoltRegProt_Q	:=	S_SPI_MNG_94.Digital_Feedback_Q	;
S_SPI_MNG_95	(Digital_Feedback_Value:=	emC_LUC[LUC_Num].SCADA.Out.BmsRackTempRegProt	,TimeTag:=Timestamp,IV:=FALSE);	BmsRackTempRegProt_Q	:=	S_SPI_MNG_95.Digital_Feedback_Q	;
S_SPI_MNG_96	(Digital_Feedback_Value:=	emC_LUC[LUC_Num].SCADA.Out.BmsAuxProtProt	,TimeTag:=Timestamp,IV:=FALSE);	BmsAuxProtProt_Q	:=	S_SPI_MNG_96.Digital_Feedback_Q	;
S_SPI_MNG_97	(Digital_Feedback_Value:=	emC_LUC[LUC_Num].SCADA.Out.BmsChargeOperLimProt	,TimeTag:=Timestamp,IV:=FALSE);	BmsChargeOperLimProt_Q	:=	S_SPI_MNG_97.Digital_Feedback_Q	;
S_SPI_MNG_98	(Digital_Feedback_Value:=	emC_LUC[LUC_Num].SCADA.Out.BmsDischargeOperLimProt	,TimeTag:=Timestamp,IV:=FALSE);	BmsDischargeOperLimProt_Q	:=	S_SPI_MNG_98.Digital_Feedback_Q	;
S_SPI_MNG_99	(Digital_Feedback_Value:=	emC_LUC[LUC_Num].SCADA.Out.BmsRackUnVoltProt	,TimeTag:=Timestamp,IV:=FALSE);	BmsRackUnVoltProt_Q	:=	S_SPI_MNG_99.Digital_Feedback_Q	;
S_SPI_MNG_100	(Digital_Feedback_Value:=	emC_LUC[LUC_Num].SCADA.Out.BmsRackOvVoltProt	,TimeTag:=Timestamp,IV:=FALSE);	BmsRackOvVoltProt_Q	:=	S_SPI_MNG_100.Digital_Feedback_Q	;
S_SPI_MNG_101	(Digital_Feedback_Value:=	emC_LUC[LUC_Num].SCADA.Out.BmsRackCommsProt	,TimeTag:=Timestamp,IV:=FALSE);	BmsRackCommsProt_Q	:=	S_SPI_MNG_101.Digital_Feedback_Q	;
S_SPI_MNG_102	(Digital_Feedback_Value:=	emC_LUC[LUC_Num].SCADA.Out.BmsTrayCommsProt	,TimeTag:=Timestamp,IV:=FALSE);	BmsTrayCommsProt_Q	:=	S_SPI_MNG_102.Digital_Feedback_Q	;
S_SPI_MNG_103	(Digital_Feedback_Value:=	emC_LUC[LUC_Num].SCADA.Out.BmsDcCntrSensor1Prot	,TimeTag:=Timestamp,IV:=FALSE);	BmsDcCntrSensor1Prot_Q	:=	S_SPI_MNG_103.Digital_Feedback_Q	;
S_SPI_MNG_104	(Digital_Feedback_Value:=	emC_LUC[LUC_Num].SCADA.Out.BmsDcCntrSensor2Prot	,TimeTag:=Timestamp,IV:=FALSE);	BmsDcCntrSensor2Prot_Q	:=	S_SPI_MNG_104.Digital_Feedback_Q	;
S_SPI_MNG_105	(Digital_Feedback_Value:=	emC_LUC[LUC_Num].SCADA.Out.BmsFanFailProt	,TimeTag:=Timestamp,IV:=FALSE);	BmsFanFailProt_Q	:=	S_SPI_MNG_105.Digital_Feedback_Q	;
S_SPI_MNG_106	(Digital_Feedback_Value:=	emC_LUC[LUC_Num].SCADA.Out.BmsChargeOverCurrentProt	,TimeTag:=Timestamp,IV:=FALSE);	BmsChargeOverCurrentProt_Q	:=	S_SPI_MNG_106.Digital_Feedback_Q	;
S_SPI_MNG_107	(Digital_Feedback_Value:=	emC_LUC[LUC_Num].SCADA.Out.BmsDisChargeOverCurrentProt	,TimeTag:=Timestamp,IV:=FALSE);	BmsDisChargeOverCurrentProt_Q	:=	S_SPI_MNG_107.Digital_Feedback_Q	;
S_SPI_MNG_108	(Digital_Feedback_Value:=	emC_LUC[LUC_Num].SCADA.Out.BmsRackVSenseDiffProt	,TimeTag:=Timestamp,IV:=FALSE);	BmsRackVSenseDiffProt_Q	:=	S_SPI_MNG_108.Digital_Feedback_Q	;
S_SPI_MNG_109	(Digital_Feedback_Value:=	emC_LUC[LUC_Num].SCADA.Out.BmsRackFuseFailProt	,TimeTag:=Timestamp,IV:=FALSE);	BmsRackFuseFailProt_Q	:=	S_SPI_MNG_109.Digital_Feedback_Q	;
S_SPI_MNG_110	(Digital_Feedback_Value:=	emC_LUC[LUC_Num].SCADA.Out.BmsRackCurrentSenserFailProt	,TimeTag:=Timestamp,IV:=FALSE);	BmsRackCurrentSenserFailProt_Q	:=	S_SPI_MNG_110.Digital_Feedback_Q	;
S_SPI_MNG_111	(Digital_Feedback_Value:=	emC_LUC[LUC_Num].SCADA.Out.BmsRackPermanentUVProt	,TimeTag:=Timestamp,IV:=FALSE);	BmsRackPermanentUVProt_Q	:=	S_SPI_MNG_111.Digital_Feedback_Q	;
S_SPI_MNG_112	(Digital_Feedback_Value:=	emC_LUC[LUC_Num].SCADA.Out.BmsDcCntr1Prot	,TimeTag:=Timestamp,IV:=FALSE);	BmsDcCntr1Prot_Q	:=	S_SPI_MNG_112.Digital_Feedback_Q	;
S_SPI_MNG_113	(Digital_Feedback_Value:=	emC_LUC[LUC_Num].SCADA.Out.BmsDcCntr2Prot	,TimeTag:=Timestamp,IV:=FALSE);	BmsDcCntr2Prot_Q	:=	S_SPI_MNG_113.Digital_Feedback_Q	;
S_SPI_MNG_114	(Digital_Feedback_Value:=	emC_LUC[LUC_Num].SCADA.Out.BmsDcSwCntFailProt	,TimeTag:=Timestamp,IV:=FALSE);	BmsDcSwCntFailProt_Q	:=	S_SPI_MNG_114.Digital_Feedback_Q	;
S_SPI_MNG_115	(Digital_Feedback_Value:=	emC_LUC[LUC_Num].SCADA.Out.BmsCellVoltSenFailProt	,TimeTag:=Timestamp,IV:=FALSE);	BmsCellVoltSenFailProt_Q	:=	S_SPI_MNG_115.Digital_Feedback_Q	;
S_SPI_MNG_116	(Digital_Feedback_Value:=	emC_LUC[LUC_Num].SCADA.Out.BmsDCFuseSenserFailProt	,TimeTag:=Timestamp,IV:=FALSE);	BmsDCFuseSenserFailProt_Q	:=	S_SPI_MNG_116.Digital_Feedback_Q	;
								
								
								
S_SPI_MNG_117	(Digital_Feedback_Value:=	emC_LUC[LUC_Num].SCADA.Out.GCRunningSt	,TimeTag:=Timestamp,IV:=FALSE);	GCRunningSt_Q	:=	S_SPI_MNG_117.Digital_Feedback_Q	;
S_SPI_MNG_118	(Digital_Feedback_Value:=	emC_LUC[LUC_Num].SCADA.Out.GCHealthy	,TimeTag:=Timestamp,IV:=FALSE);	GCHealthy_Q	:=	S_SPI_MNG_118.Digital_Feedback_Q	;
S_SPI_MNG_119	(Digital_Feedback_Value:=	emC_LUC[LUC_Num].SCADA.Out.GCStartingSt	,TimeTag:=Timestamp,IV:=FALSE);	GCStartingSt_Q	:=	S_SPI_MNG_119.Digital_Feedback_Q	;
S_SPI_MNG_120	(Digital_Feedback_Value:=	emC_LUC[LUC_Num].SCADA.Out.GCReadySt	,TimeTag:=Timestamp,IV:=FALSE);	GCReadySt_Q	:=	S_SPI_MNG_120.Digital_Feedback_Q	;
S_SPI_MNG_121	(Digital_Feedback_Value:=	emC_LUC[LUC_Num].SCADA.Out.GCGridFollowing	,TimeTag:=Timestamp,IV:=FALSE);	GCGridFollowing_Q	:=	S_SPI_MNG_121.Digital_Feedback_Q	;
S_SPI_MNG_122	(Digital_Feedback_Value:=	emC_LUC[LUC_Num].SCADA.Out.GCFaultSt	,TimeTag:=Timestamp,IV:=FALSE);	GCFaultSt_Q	:=	S_SPI_MNG_122.Digital_Feedback_Q	;
S_SPI_MNG_123	(Digital_Feedback_Value:=	emC_LUC[LUC_Num].SCADA.Out.GCGridForming	,TimeTag:=Timestamp,IV:=FALSE);	GCGridForming_Q	:=	S_SPI_MNG_123.Digital_Feedback_Q	;
S_SPI_MNG_124	(Digital_Feedback_Value:=	emC_LUC[LUC_Num].SCADA.Out.GCAreaEPSLost	,TimeTag:=Timestamp,IV:=FALSE);	GCAreaEPSLost_Q	:=	S_SPI_MNG_124.Digital_Feedback_Q	;
S_SPI_MNG_125	(Digital_Feedback_Value:=	emC_LUC[LUC_Num].SCADA.Out.GCChargingSt	,TimeTag:=Timestamp,IV:=FALSE);	GCChargingSt_Q	:=	S_SPI_MNG_125.Digital_Feedback_Q	;
S_SPI_MNG_126	(Digital_Feedback_Value:=	emC_LUC[LUC_Num].SCADA.Out.GCRideThru	,TimeTag:=Timestamp,IV:=FALSE);	GCRideThru_Q	:=	S_SPI_MNG_126.Digital_Feedback_Q	;
S_SPI_MNG_127	(Digital_Feedback_Value:=	emC_LUC[LUC_Num].SCADA.Out.GCTransitionActiveSt	,TimeTag:=Timestamp,IV:=FALSE);	GCTransitionActiveSt_Q	:=	S_SPI_MNG_127.Digital_Feedback_Q	;
S_SPI_MNG_128	(Digital_Feedback_Value:=	emC_LUC[LUC_Num].SCADA.Out.GCGndFault	,TimeTag:=Timestamp,IV:=FALSE);	GCGndFault_Q	:=	S_SPI_MNG_128.Digital_Feedback_Q	;
S_SPI_MNG_129	(Digital_Feedback_Value:=	emC_LUC[LUC_Num].SCADA.Out.GCDCOverU	,TimeTag:=Timestamp,IV:=FALSE);	GCDCOverU_Q	:=	S_SPI_MNG_129.Digital_Feedback_Q	;
S_SPI_MNG_130	(Digital_Feedback_Value:=	emC_LUC[LUC_Num].SCADA.Out.GCACDisconnect	,TimeTag:=Timestamp,IV:=FALSE);	GCACDisconnect_Q	:=	S_SPI_MNG_130.Digital_Feedback_Q	;
S_SPI_MNG_131	(Digital_Feedback_Value:=	emC_LUC[LUC_Num].SCADA.Out.GCDCDisconnect	,TimeTag:=Timestamp,IV:=FALSE);	GCDCDisconnect_Q	:=	S_SPI_MNG_131.Digital_Feedback_Q	;
S_SPI_MNG_132	(Digital_Feedback_Value:=	emC_LUC[LUC_Num].SCADA.Out.GCDCGridDisconnect	,TimeTag:=Timestamp,IV:=FALSE);	GCDCGridDisconnect_Q	:=	S_SPI_MNG_132.Digital_Feedback_Q	;
S_SPI_MNG_133	(Digital_Feedback_Value:=	emC_LUC[LUC_Num].SCADA.Out.GCCabinetOpen	,TimeTag:=Timestamp,IV:=FALSE);	GCCabinetOpen_Q	:=	S_SPI_MNG_133.Digital_Feedback_Q	;
S_SPI_MNG_134	(Digital_Feedback_Value:=	emC_LUC[LUC_Num].SCADA.Out.GCManualShutdown	,TimeTag:=Timestamp,IV:=FALSE);	GCManualShutdown_Q	:=	S_SPI_MNG_134.Digital_Feedback_Q	;
S_SPI_MNG_135	(Digital_Feedback_Value:=	emC_LUC[LUC_Num].SCADA.Out.GCOverTemp	,TimeTag:=Timestamp,IV:=FALSE);	GCOverTemp_Q	:=	S_SPI_MNG_135.Digital_Feedback_Q	;
S_SPI_MNG_136	(Digital_Feedback_Value:=	emC_LUC[LUC_Num].SCADA.Out.GCOverF	,TimeTag:=Timestamp,IV:=FALSE);	GCOverF_Q	:=	S_SPI_MNG_136.Digital_Feedback_Q	;
S_SPI_MNG_137	(Digital_Feedback_Value:=	emC_LUC[LUC_Num].SCADA.Out.GCUnderF	,TimeTag:=Timestamp,IV:=FALSE);	GCUnderF_Q	:=	S_SPI_MNG_137.Digital_Feedback_Q	;
S_SPI_MNG_138	(Digital_Feedback_Value:=	emC_LUC[LUC_Num].SCADA.Out.GCACOverVolt	,TimeTag:=Timestamp,IV:=FALSE);	GCACOverVolt_Q	:=	S_SPI_MNG_138.Digital_Feedback_Q	;
S_SPI_MNG_139	(Digital_Feedback_Value:=	emC_LUC[LUC_Num].SCADA.Out.GCACUnderVolt	,TimeTag:=Timestamp,IV:=FALSE);	GCACUnderVolt_Q	:=	S_SPI_MNG_139.Digital_Feedback_Q	;
S_SPI_MNG_140	(Digital_Feedback_Value:=	emC_LUC[LUC_Num].SCADA.Out.GCBlownFuse	,TimeTag:=Timestamp,IV:=FALSE);	GCBlownFuse_Q	:=	S_SPI_MNG_140.Digital_Feedback_Q	;
S_SPI_MNG_141	(Digital_Feedback_Value:=	emC_LUC[LUC_Num].SCADA.Out.GCUnderTemp	,TimeTag:=Timestamp,IV:=FALSE);	GCUnderTemp_Q	:=	S_SPI_MNG_141.Digital_Feedback_Q	;
S_SPI_MNG_142	(Digital_Feedback_Value:=	emC_LUC[LUC_Num].SCADA.Out.GCMemLoss	,TimeTag:=Timestamp,IV:=FALSE);	GCMemLoss_Q	:=	S_SPI_MNG_142.Digital_Feedback_Q	;
S_SPI_MNG_143	(Digital_Feedback_Value:=	emC_LUC[LUC_Num].SCADA.Out.GCHWTestFailed	,TimeTag:=Timestamp,IV:=FALSE);	GCHWTestFailed_Q	:=	S_SPI_MNG_143.Digital_Feedback_Q	;
S_SPI_MNG_162	(Digital_Feedback_Value:=	emC_LUC[LUC_Num].SCADA.Out.GCABBCtrlWrongConfig	,TimeTag:=Timestamp,IV:=FALSE);	GCABBCtrlWrongConfig_Q	:=	S_SPI_MNG_162.Digital_Feedback_Q	;
S_SPI_MNG_163	(Digital_Feedback_Value:=	emC_LUC[LUC_Num].SCADA.Out.GCABBCtrlReady	,TimeTag:=Timestamp,IV:=FALSE);	GCABBCtrlReady_Q	:=	S_SPI_MNG_163.Digital_Feedback_Q	;
S_SPI_MNG_164	(Digital_Feedback_Value:=	emC_LUC[LUC_Num].SCADA.Out.GCABBCtrlStartingSt	,TimeTag:=Timestamp,IV:=FALSE);	GCABBCtrlStartingSt_Q	:=	S_SPI_MNG_164.Digital_Feedback_Q	;
S_SPI_MNG_165	(Digital_Feedback_Value:=	emC_LUC[LUC_Num].SCADA.Out.GCABBCtrlVGMActiveSt	,TimeTag:=Timestamp,IV:=FALSE);	GCABBCtrlVGMActiveSt_Q	:=	S_SPI_MNG_165.Digital_Feedback_Q	;
S_SPI_MNG_166	(Digital_Feedback_Value:=	emC_LUC[LUC_Num].SCADA.Out.GCABBCtrlGSMActiveSt	,TimeTag:=Timestamp,IV:=FALSE);	GCABBCtrlGSMActiveSt_Q	:=	S_SPI_MNG_166.Digital_Feedback_Q	;
S_SPI_MNG_167	(Digital_Feedback_Value:=	emC_LUC[LUC_Num].SCADA.Out.GCABBCtrlError	,TimeTag:=Timestamp,IV:=FALSE);	GCABBCtrlError_Q	:=	S_SPI_MNG_167.Digital_Feedback_Q	;
S_SPI_MNG_168	(Digital_Feedback_Value:=	emC_LUC[LUC_Num].SCADA.Out.GCABBCtrlStoppingSt	,TimeTag:=Timestamp,IV:=FALSE);	GCABBCtrlStoppingSt_Q	:=	S_SPI_MNG_168.Digital_Feedback_Q	;
S_SPI_MNG_169	(Digital_Feedback_Value:=	emC_LUC[LUC_Num].SCADA.Out.GCABBCtrlIslanded	,TimeTag:=Timestamp,IV:=FALSE);	GCABBCtrlIslanded_Q	:=	S_SPI_MNG_169.Digital_Feedback_Q	;
S_SPI_MNG_172	(Digital_Feedback_Value:=	emC_LUC[LUC_Num].SCADA.Out.GCLostComms	,TimeTag:=Timestamp,IV:=FALSE);	GCLostComms_Q	:=	S_SPI_MNG_172.Digital_Feedback_Q	;
S_SPI_MNG_173	(Digital_Feedback_Value:=	emC_LUC[LUC_Num].SCADA.Out.GCCommsOk	,TimeTag:=Timestamp,IV:=FALSE);	GCCommsOk_Q	:=	S_SPI_MNG_173.Digital_Feedback_Q	;
S_SPI_MNG_174	(Digital_Feedback_Value:=	emC_LUC[LUC_Num].SCADA.Out.GCHardwareenablestatus	,TimeTag:=Timestamp,IV:=FALSE);	GCHardwareenablestatus_Q	:=	S_SPI_MNG_174.Digital_Feedback_Q	;
S_SPI_MNG_175	(Digital_Feedback_Value:=	emC_LUC[LUC_Num].SCADA.Out.GCACPowerAvailable	,TimeTag:=Timestamp,IV:=FALSE);	GCACPowerAvailable_Q	:=	S_SPI_MNG_175.Digital_Feedback_Q	;
S_SPI_MNG_176	(Digital_Feedback_Value:=	emC_LUC[LUC_Num].SCADA.Out.GCDCPowerAvailable	,TimeTag:=Timestamp,IV:=FALSE);	GCDCPowerAvailable_Q	:=	S_SPI_MNG_176.Digital_Feedback_Q	;
S_SPI_MNG_177	(Digital_Feedback_Value:=	emC_LUC[LUC_Num].SCADA.Out.GCPowerCircuitEnabled	,TimeTag:=Timestamp,IV:=FALSE);	GCPowerCircuitEnabled_Q	:=	S_SPI_MNG_177.Digital_Feedback_Q	;
S_SPI_MNG_178	(Digital_Feedback_Value:=	emC_LUC[LUC_Num].SCADA.Out.GCMX1relaystatus	,TimeTag:=Timestamp,IV:=FALSE);	GCMX1relaystatus_Q	:=	S_SPI_MNG_178.Digital_Feedback_Q	;
S_SPI_MNG_179	(Digital_Feedback_Value:=	emC_LUC[LUC_Num].SCADA.Out.GCMX2relaystatus	,TimeTag:=Timestamp,IV:=FALSE);	GCMX2relaystatus_Q	:=	S_SPI_MNG_179.Digital_Feedback_Q	;
S_SPI_MNG_180	(Digital_Feedback_Value:=	emC_LUC[LUC_Num].SCADA.Out.GCPrechargestatus	,TimeTag:=Timestamp,IV:=FALSE);	GCPrechargestatus_Q	:=	S_SPI_MNG_180.Digital_Feedback_Q	;
S_SPI_MNG_181	(Digital_Feedback_Value:=	emC_LUC[LUC_Num].SCADA.Out.GCK2Relaystatus	,TimeTag:=Timestamp,IV:=FALSE);	GCK2Relaystatus_Q	:=	S_SPI_MNG_181.Digital_Feedback_Q	;
S_SPI_MNG_182	(Digital_Feedback_Value:=	emC_LUC[LUC_Num].SCADA.Out.GCControlcommandsvalid	,TimeTag:=Timestamp,IV:=FALSE);	GCControlcommandsvalid_Q	:=	S_SPI_MNG_182.Digital_Feedback_Q	;
S_SPI_MNG_183	(Digital_Feedback_Value:=	emC_LUC[LUC_Num].SCADA.Out.GCPowercommandValid	,TimeTag:=Timestamp,IV:=FALSE);	GCPowercommandValid_Q	:=	S_SPI_MNG_183.Digital_Feedback_Q	;
S_SPI_MNG_184	(Digital_Feedback_Value:=	emC_LUC[LUC_Num].SCADA.Out.GCCurrentcommandValid	,TimeTag:=Timestamp,IV:=FALSE);	GCCurrentcommandValid_Q	:=	S_SPI_MNG_184.Digital_Feedback_Q	;
S_SPI_MNG_185	(Digital_Feedback_Value:=	emC_LUC[LUC_Num].SCADA.Out.GCPhaserotationstatus	,TimeTag:=Timestamp,IV:=FALSE);	GCPhaserotationstatus_Q	:=	S_SPI_MNG_185.Digital_Feedback_Q	;
S_SPI_MNG_186	(Digital_Feedback_Value:=	emC_LUC[LUC_Num].SCADA.Out.GCLinevoltagedetected	,TimeTag:=Timestamp,IV:=FALSE);	GCLinevoltagedetected_Q	:=	S_SPI_MNG_186.Digital_Feedback_Q	;
S_SPI_MNG_187	(Digital_Feedback_Value:=	emC_LUC[LUC_Num].SCADA.Out.GCUnused	,TimeTag:=Timestamp,IV:=FALSE);	GCUnused_Q	:=	S_SPI_MNG_187.Digital_Feedback_Q	;
S_SPI_MNG_188	(Digital_Feedback_Value:=	emC_LUC[LUC_Num].SCADA.Out.GCRemoteACPowerAvailable	,TimeTag:=Timestamp,IV:=FALSE);	GCRemoteACPowerAvailable_Q	:=	S_SPI_MNG_188.Digital_Feedback_Q	;
S_SPI_MNG_189	(Digital_Feedback_Value:=	emC_LUC[LUC_Num].SCADA.Out.GCRemotephaserotationstatus	,TimeTag:=Timestamp,IV:=FALSE);	GCRemotephaserotationstatus_Q	:=	S_SPI_MNG_189.Digital_Feedback_Q	;
S_SPI_MNG_190	(Digital_Feedback_Value:=	emC_LUC[LUC_Num].SCADA.Out.GCRemoteLineVoltageDetected	,TimeTag:=Timestamp,IV:=FALSE);	GCRemoteLineVoltageDetected_Q	:=	S_SPI_MNG_190.Digital_Feedback_Q	;
S_SPI_MNG_191	(Digital_Feedback_Value:=	emC_LUC[LUC_Num].SCADA.Out.GCDI1Status	,TimeTag:=Timestamp,IV:=FALSE);	GCDI1Status_Q	:=	S_SPI_MNG_191.Digital_Feedback_Q	;
S_SPI_MNG_192	(Digital_Feedback_Value:=	emC_LUC[LUC_Num].SCADA.Out.GCDI2Status	,TimeTag:=Timestamp,IV:=FALSE);	GCDI2Status_Q	:=	S_SPI_MNG_192.Digital_Feedback_Q	;
S_SPI_MNG_193	(Digital_Feedback_Value:=	emC_LUC[LUC_Num].SCADA.Out.GCDI3Status	,TimeTag:=Timestamp,IV:=FALSE);	GCDI3Status_Q	:=	S_SPI_MNG_193.Digital_Feedback_Q	;
S_SPI_MNG_194	(Digital_Feedback_Value:=	emC_LUC[LUC_Num].SCADA.Out.GCDI4Status	,TimeTag:=Timestamp,IV:=FALSE);	GCDI4Status_Q	:=	S_SPI_MNG_194.Digital_Feedback_Q	;
S_SPI_MNG_195	(Digital_Feedback_Value:=	emC_LUC[LUC_Num].SCADA.Out.GCDO1Status	,TimeTag:=Timestamp,IV:=FALSE);	GCDO1Status_Q	:=	S_SPI_MNG_195.Digital_Feedback_Q	;
S_SPI_MNG_196	(Digital_Feedback_Value:=	emC_LUC[LUC_Num].SCADA.Out.GCDO2Status	,TimeTag:=Timestamp,IV:=FALSE);	GCDO2Status_Q	:=	S_SPI_MNG_196.Digital_Feedback_Q	;
S_SPI_MNG_197	(Digital_Feedback_Value:=	emC_LUC[LUC_Num].SCADA.Out.GCDO3Status	,TimeTag:=Timestamp,IV:=FALSE);	GCDO3Status_Q	:=	S_SPI_MNG_197.Digital_Feedback_Q	;
S_SPI_MNG_198	(Digital_Feedback_Value:=	emC_LUC[LUC_Num].SCADA.Out.GCDO4Status	,TimeTag:=Timestamp,IV:=FALSE);	GCDO4Status_Q	:=	S_SPI_MNG_198.Digital_Feedback_Q	;
S_SPI_MNG_199	(Digital_Feedback_Value:=	emC_LUC[LUC_Num].SCADA.Out.GCDClinkRefCmdValid	,TimeTag:=Timestamp,IV:=FALSE);	GCDClinkRefCmdValid_Q	:=	S_SPI_MNG_199.Digital_Feedback_Q	;
S_SPI_MNG_200	(Digital_Feedback_Value:=	emC_LUC[LUC_Num].SCADA.Out.GCPumpRunning	,TimeTag:=Timestamp,IV:=FALSE);	GCPumpRunning_Q	:=	S_SPI_MNG_200.Digital_Feedback_Q	;
S_SPI_MNG_201	(Digital_Feedback_Value:=	emC_LUC[LUC_Num].SCADA.Out.GCPumpFault	,TimeTag:=Timestamp,IV:=FALSE);	GCPumpFault_Q	:=	S_SPI_MNG_201.Digital_Feedback_Q	;
S_SPI_MNG_202	(Digital_Feedback_Value:=	emC_LUC[LUC_Num].SCADA.Out.GCABBLostCommsStop	,TimeTag:=Timestamp,IV:=FALSE);	GCABBLostCommsStop_Q	:=	S_SPI_MNG_202.Digital_Feedback_Q	;
S_SPI_MNG_203	(Digital_Feedback_Value:=	emC_LUC[LUC_Num].SCADA.Out.GCCtrlSystemReady	,TimeTag:=Timestamp,IV:=FALSE);	CtrlSystemReady_Q	:=	S_SPI_MNG_203.Digital_Feedback_Q	;
S_SPI_MNG_205	(Digital_Feedback_Value:=	emC_LUC[LUC_Num].SCADA.Out.GCFlt_Estp	,TimeTag:=Timestamp,IV:=FALSE);	GCFlt_Estp_Q	:=	S_SPI_MNG_205.Digital_Feedback_Q	;
S_SPI_MNG_206	(Digital_Feedback_Value:=	emC_LUC[LUC_Num].SCADA.Out.GCFlt_ACOverCurrent	,TimeTag:=Timestamp,IV:=FALSE);	GCFlt_ACOverCurrent_Q	:=	S_SPI_MNG_206.Digital_Feedback_Q	;
S_SPI_MNG_207	(Digital_Feedback_Value:=	emC_LUC[LUC_Num].SCADA.Out.GCFlt_DCOverCurrent	,TimeTag:=Timestamp,IV:=FALSE);	GCFlt_DCOverCurrent_Q	:=	S_SPI_MNG_207.Digital_Feedback_Q	;
S_SPI_MNG_208	(Digital_Feedback_Value:=	emC_LUC[LUC_Num].SCADA.Out.GCFlt_DCOverVoltage	,TimeTag:=Timestamp,IV:=FALSE);	GCFlt_DCOverVoltage_Q	:=	S_SPI_MNG_208.Digital_Feedback_Q	;
S_SPI_MNG_209	(Digital_Feedback_Value:=	emC_LUC[LUC_Num].SCADA.Out.GCFlt_PDOverTemp	,TimeTag:=Timestamp,IV:=FALSE);	GCFlt_PDOverTemp_Q	:=	S_SPI_MNG_209.Digital_Feedback_Q	;
S_SPI_MNG_210	(Digital_Feedback_Value:=	emC_LUC[LUC_Num].SCADA.Out.GCFlt_InvOverTemp	,TimeTag:=Timestamp,IV:=FALSE);	GCFlt_InvOverTemp_Q	:=	S_SPI_MNG_210.Digital_Feedback_Q	;
S_SPI_MNG_211	(Digital_Feedback_Value:=	emC_LUC[LUC_Num].SCADA.Out.GCFlt_CmdMsg	,TimeTag:=Timestamp,IV:=FALSE);	GCFlt_CmdMsg_Q	:=	S_SPI_MNG_211.Digital_Feedback_Q	;
S_SPI_MNG_212	(Digital_Feedback_Value:=	emC_LUC[LUC_Num].SCADA.Out.GCFlt_DCUnderVolt	,TimeTag:=Timestamp,IV:=FALSE);	GCFlt_DCUnderVolt_Q	:=	S_SPI_MNG_212.Digital_Feedback_Q	;
S_SPI_MNG_213	(Digital_Feedback_Value:=	emC_LUC[LUC_Num].SCADA.Out.GCFlt_ACOverVolt	,TimeTag:=Timestamp,IV:=FALSE);	GCFlt_ACOverVolt_Q	:=	S_SPI_MNG_213.Digital_Feedback_Q	;
S_SPI_MNG_214	(Digital_Feedback_Value:=	emC_LUC[LUC_Num].SCADA.Out.GCFlt_IllegalTrans	,TimeTag:=Timestamp,IV:=FALSE);	GCFlt_IllegalTrans_Q	:=	S_SPI_MNG_214.Digital_Feedback_Q	;
S_SPI_MNG_215	(Digital_Feedback_Value:=	emC_LUC[LUC_Num].SCADA.Out.GCFlt_EEHeat	,TimeTag:=Timestamp,IV:=FALSE);	GCFlt_EEHeat_Q	:=	S_SPI_MNG_215.Digital_Feedback_Q	;
S_SPI_MNG_216	(Digital_Feedback_Value:=	emC_LUC[LUC_Num].SCADA.Out.GCFlt_EESction	,TimeTag:=Timestamp,IV:=FALSE);	GCFlt_EESction_Q	:=	S_SPI_MNG_216.Digital_Feedback_Q	;
S_SPI_MNG_217	(Digital_Feedback_Value:=	emC_LUC[LUC_Num].SCADA.Out.GCFlt_Cool	,TimeTag:=Timestamp,IV:=FALSE);	GCFlt_Cool_Q	:=	S_SPI_MNG_217.Digital_Feedback_Q	;
S_SPI_MNG_218	(Digital_Feedback_Value:=	emC_LUC[LUC_Num].SCADA.Out.GCFlt_TimedOverLoadAC	,TimeTag:=Timestamp,IV:=FALSE);	GCFlt_TimedOverLoadAC_Q	:=	S_SPI_MNG_218.Digital_Feedback_Q	;
S_SPI_MNG_219	(Digital_Feedback_Value:=	emC_LUC[LUC_Num].SCADA.Out.GCFlt_TimedOverLoadDC	,TimeTag:=Timestamp,IV:=FALSE);	GCFlt_TimedOverLoadDC_Q	:=	S_SPI_MNG_219.Digital_Feedback_Q	;
S_SPI_MNG_220	(Digital_Feedback_Value:=	emC_LUC[LUC_Num].SCADA.Out.GCFlt_ICOL	,TimeTag:=Timestamp,IV:=FALSE);	GCFlt_ICOL_Q	:=	S_SPI_MNG_220.Digital_Feedback_Q	;
S_SPI_MNG_221	(Digital_Feedback_Value:=	emC_LUC[LUC_Num].SCADA.Out.GCFlt_CtlBdVolt	,TimeTag:=Timestamp,IV:=FALSE);	GCFlt_CtlBdVolt_Q	:=	S_SPI_MNG_221.Digital_Feedback_Q	;
S_SPI_MNG_222	(Digital_Feedback_Value:=	emC_LUC[LUC_Num].SCADA.Out.GCFlt_PChImbal	,TimeTag:=Timestamp,IV:=FALSE);	GCFlt_PChImbal_Q	:=	S_SPI_MNG_222.Digital_Feedback_Q	;
S_SPI_MNG_223	(Digital_Feedback_Value:=	emC_LUC[LUC_Num].SCADA.Out.GCFlt_DiDt	,TimeTag:=Timestamp,IV:=FALSE);	GCFlt_DiDt_Q	:=	S_SPI_MNG_223.Digital_Feedback_Q	;
S_SPI_MNG_224	(Digital_Feedback_Value:=	emC_LUC[LUC_Num].SCADA.Out.GCFlt_CoolingFlw	,TimeTag:=Timestamp,IV:=FALSE);	GCFlt_CoolingFlw_Q	:=	S_SPI_MNG_224.Digital_Feedback_Q	;
S_SPI_MNG_225	(Digital_Feedback_Value:=	emC_LUC[LUC_Num].SCADA.Out.GCFlt_ThrmOverLoad	,TimeTag:=Timestamp,IV:=FALSE);	GCFlt_ThrmOverLoad_Q	:=	S_SPI_MNG_225.Digital_Feedback_Q	;
S_SPI_MNG_226	(Digital_Feedback_Value:=	emC_LUC[LUC_Num].SCADA.Out.GCFlt_Fan	,TimeTag:=Timestamp,IV:=FALSE);	GCFlt_Fan_Q	:=	S_SPI_MNG_226.Digital_Feedback_Q	;
S_SPI_MNG_227	(Digital_Feedback_Value:=	emC_LUC[LUC_Num].SCADA.Out.GCFlt_POR	,TimeTag:=Timestamp,IV:=FALSE);	GCFlt_POR_Q	:=	S_SPI_MNG_227.Digital_Feedback_Q	;
S_SPI_MNG_228	(Digital_Feedback_Value:=	emC_LUC[LUC_Num].SCADA.Out.GCFlt_Condensation	,TimeTag:=Timestamp,IV:=FALSE);	GCFlt_Condensation_Q	:=	S_SPI_MNG_228.Digital_Feedback_Q	;
S_SPI_MNG_229	(Digital_Feedback_Value:=	emC_LUC[LUC_Num].SCADA.Out.GCFlt_I2C	,TimeTag:=Timestamp,IV:=FALSE);	GCFlt_I2C_Q	:=	S_SPI_MNG_229.Digital_Feedback_Q	;
S_SPI_MNG_230	(Digital_Feedback_Value:=	emC_LUC[LUC_Num].SCADA.Out.GCFlt_ExternalInhibit	,TimeTag:=Timestamp,IV:=FALSE);	GCFlt_ExternalInhibit_Q	:=	S_SPI_MNG_230.Digital_Feedback_Q	;
S_SPI_MNG_231	(Digital_Feedback_Value:=	emC_LUC[LUC_Num].SCADA.Out.GCFlt_GroundFault	,TimeTag:=Timestamp,IV:=FALSE);	GCFlt_GroundFault_Q	:=	S_SPI_MNG_231.Digital_Feedback_Q	;
S_SPI_MNG_232	(Digital_Feedback_Value:=	emC_LUC[LUC_Num].SCADA.Out.GCFlt_Fuse	,TimeTag:=Timestamp,IV:=FALSE);	GCFlt_Fuse_Q	:=	S_SPI_MNG_232.Digital_Feedback_Q	;
S_SPI_MNG_233	(Digital_Feedback_Value:=	emC_LUC[LUC_Num].SCADA.Out.GCFlt_Rsvd28	,TimeTag:=Timestamp,IV:=FALSE);	GCFlt_Rsvd28_Q	:=	S_SPI_MNG_233.Digital_Feedback_Q	;
S_SPI_MNG_234	(Digital_Feedback_Value:=	emC_LUC[LUC_Num].SCADA.Out.GCFlt_ACDisconnect	,TimeTag:=Timestamp,IV:=FALSE);	GCFlt_ACDisconnect_Q	:=	S_SPI_MNG_234.Digital_Feedback_Q	;
S_SPI_MNG_235	(Digital_Feedback_Value:=	emC_LUC[LUC_Num].SCADA.Out.GCFlt_Rsvd30	,TimeTag:=Timestamp,IV:=FALSE);	GCFlt_Rsvd30_Q	:=	S_SPI_MNG_235.Digital_Feedback_Q	;
S_SPI_MNG_236	(Digital_Feedback_Value:=	emC_LUC[LUC_Num].SCADA.Out.GCFlt_Rsvd31	,TimeTag:=Timestamp,IV:=FALSE);	GCFlt_Rsvd31_Q	:=	S_SPI_MNG_236.Digital_Feedback_Q	;
S_SPI_MNG_237	(Digital_Feedback_Value:=	emC_LUC[LUC_Num].SCADA.Out.GCWrn_CANW	,TimeTag:=Timestamp,IV:=FALSE);	GCWrn_CANW_Q	:=	S_SPI_MNG_237.Digital_Feedback_Q	;
S_SPI_MNG_238	(Digital_Feedback_Value:=	emC_LUC[LUC_Num].SCADA.Out.GCWrn_CANEP	,TimeTag:=Timestamp,IV:=FALSE);	GCWrn_CANEP_Q	:=	S_SPI_MNG_238.Digital_Feedback_Q	;
S_SPI_MNG_239	(Digital_Feedback_Value:=	emC_LUC[LUC_Num].SCADA.Out.GCWrn_Thrm	,TimeTag:=Timestamp,IV:=FALSE);	GCWrn_Thrm_Q	:=	S_SPI_MNG_239.Digital_Feedback_Q	;
S_SPI_MNG_240	(Digital_Feedback_Value:=	emC_LUC[LUC_Num].SCADA.Out.GCWrn_Fan	,TimeTag:=Timestamp,IV:=FALSE);	GCWrn_Fan_Q	:=	S_SPI_MNG_240.Digital_Feedback_Q	;
S_SPI_MNG_241	(Digital_Feedback_Value:=	emC_LUC[LUC_Num].SCADA.Out.GCWrn_EeSaveActive	,TimeTag:=Timestamp,IV:=FALSE);	GCWrn_EeSaveActive_Q	:=	S_SPI_MNG_241.Digital_Feedback_Q	;
S_SPI_MNG_242	(Digital_Feedback_Value:=	emC_LUC[LUC_Num].SCADA.Out.GCWrn_LocNetMismatch	,TimeTag:=Timestamp,IV:=FALSE);	GCWrn_LocNetMismatch_Q	:=	S_SPI_MNG_242.Digital_Feedback_Q	;
S_SPI_MNG_243	(Digital_Feedback_Value:=	emC_LUC[LUC_Num].SCADA.Out.GCWrn_RemNetMismatch	,TimeTag:=Timestamp,IV:=FALSE);	GCWrn_RemNetMismatch_Q	:=	S_SPI_MNG_243.Digital_Feedback_Q	;
S_SPI_MNG_244	(Digital_Feedback_Value:=	emC_LUC[LUC_Num].SCADA.Out.GCWrn_Condensation	,TimeTag:=Timestamp,IV:=FALSE);	GCWrn_Condensation_Q	:=	S_SPI_MNG_244.Digital_Feedback_Q	;
S_SPI_MNG_245	(Digital_Feedback_Value:=	emC_LUC[LUC_Num].SCADA.Out.GCWrn_I2C	,TimeTag:=Timestamp,IV:=FALSE);	GCWrn_I2C_Q	:=	S_SPI_MNG_245.Digital_Feedback_Q	;
S_SPI_MNG_246	(Digital_Feedback_Value:=	emC_LUC[LUC_Num].SCADA.Out.GCWrn_ExternalInhibit	,TimeTag:=Timestamp,IV:=FALSE);	GCWrn_ExternalInhibit_Q	:=	S_SPI_MNG_246.Digital_Feedback_Q	;
S_SPI_MNG_247	(Digital_Feedback_Value:=	emC_LUC[LUC_Num].SCADA.Out.GCWrn_MaintReqd	,TimeTag:=Timestamp,IV:=FALSE);	GCWrn_MaintReqd_Q	:=	S_SPI_MNG_247.Digital_Feedback_Q	;
S_SPI_MNG_248	(Digital_Feedback_Value:=	emC_LUC[LUC_Num].SCADA.Out.GCWrn_GroundFault	,TimeTag:=Timestamp,IV:=FALSE);	GCWrn_GroundFault_Q	:=	S_SPI_MNG_248.Digital_Feedback_Q	;
S_SPI_MNG_249	(Digital_Feedback_Value:=	emC_LUC[LUC_Num].SCADA.Out.GCWrn_Fuse	,TimeTag:=Timestamp,IV:=FALSE);	GCWrn_Fuse_Q	:=	S_SPI_MNG_249.Digital_Feedback_Q	;
S_SPI_MNG_250	(Digital_Feedback_Value:=	emC_LUC[LUC_Num].SCADA.Out.GCWrn_ACDisconnect	,TimeTag:=Timestamp,IV:=FALSE);	GCWrn_ACDisconnect_Q	:=	S_SPI_MNG_250.Digital_Feedback_Q	;
S_SPI_MNG_251	(Digital_Feedback_Value:=	emC_LUC[LUC_Num].SCADA.Out.GCWrn_Rsvd14	,TimeTag:=Timestamp,IV:=FALSE);	GCWrn_Rsvd14_Q	:=	S_SPI_MNG_251.Digital_Feedback_Q	;
S_SPI_MNG_252	(Digital_Feedback_Value:=	emC_LUC[LUC_Num].SCADA.Out.GCWrn_Rsvd15	,TimeTag:=Timestamp,IV:=FALSE);	GCWrn_Rsvd15_Q	:=	S_SPI_MNG_252.Digital_Feedback_Q	;
S_SPI_MNG_253	(Digital_Feedback_Value:=	emC_LUC[LUC_Num].SCADA.Out.GCWrn_Rsvd16	,TimeTag:=Timestamp,IV:=FALSE);	GCWrn_Rsvd16_Q	:=	S_SPI_MNG_253.Digital_Feedback_Q	;
S_SPI_MNG_254	(Digital_Feedback_Value:=	emC_LUC[LUC_Num].SCADA.Out.GCWrn_Rsvd17	,TimeTag:=Timestamp,IV:=FALSE);	GCWrn_Rsvd17_Q	:=	S_SPI_MNG_254.Digital_Feedback_Q	;
S_SPI_MNG_255	(Digital_Feedback_Value:=	emC_LUC[LUC_Num].SCADA.Out.GCWrn_Rsvd18	,TimeTag:=Timestamp,IV:=FALSE);	GCWrn_Rsvd18_Q	:=	S_SPI_MNG_255.Digital_Feedback_Q	;
S_SPI_MNG_256	(Digital_Feedback_Value:=	emC_LUC[LUC_Num].SCADA.Out.GCWrn_Rsvd19	,TimeTag:=Timestamp,IV:=FALSE);	GCWrn_Rsvd19_Q	:=	S_SPI_MNG_256.Digital_Feedback_Q	;
S_SPI_MNG_257	(Digital_Feedback_Value:=	emC_LUC[LUC_Num].SCADA.Out.GCWrn_Rsvd20	,TimeTag:=Timestamp,IV:=FALSE);	GCWrn_Rsvd20_Q	:=	S_SPI_MNG_257.Digital_Feedback_Q	;
S_SPI_MNG_258	(Digital_Feedback_Value:=	emC_LUC[LUC_Num].SCADA.Out.GCWrn_Rsvd21	,TimeTag:=Timestamp,IV:=FALSE);	GCWrn_Rsvd21_Q	:=	S_SPI_MNG_258.Digital_Feedback_Q	;
S_SPI_MNG_259	(Digital_Feedback_Value:=	emC_LUC[LUC_Num].SCADA.Out.GCWrn_Rsvd22	,TimeTag:=Timestamp,IV:=FALSE);	GCWrn_Rsvd22_Q	:=	S_SPI_MNG_259.Digital_Feedback_Q	;
S_SPI_MNG_260	(Digital_Feedback_Value:=	emC_LUC[LUC_Num].SCADA.Out.GCWrn_Rsvd23	,TimeTag:=Timestamp,IV:=FALSE);	GCWrn_Rsvd23_Q	:=	S_SPI_MNG_260.Digital_Feedback_Q	;
S_SPI_MNG_261	(Digital_Feedback_Value:=	emC_LUC[LUC_Num].SCADA.Out.GCWrn_Rsvd24	,TimeTag:=Timestamp,IV:=FALSE);	GCWrn_Rsvd24_Q	:=	S_SPI_MNG_261.Digital_Feedback_Q	;
S_SPI_MNG_262	(Digital_Feedback_Value:=	emC_LUC[LUC_Num].SCADA.Out.GCWrn_Rsvd25	,TimeTag:=Timestamp,IV:=FALSE);	GCWrn_Rsvd25_Q	:=	S_SPI_MNG_262.Digital_Feedback_Q	;
S_SPI_MNG_263	(Digital_Feedback_Value:=	emC_LUC[LUC_Num].SCADA.Out.GCWrn_Rsvd26	,TimeTag:=Timestamp,IV:=FALSE);	GCWrn_Rsvd26_Q	:=	S_SPI_MNG_263.Digital_Feedback_Q	;
S_SPI_MNG_264	(Digital_Feedback_Value:=	emC_LUC[LUC_Num].SCADA.Out.GCWrn_Rsvd27	,TimeTag:=Timestamp,IV:=FALSE);	GCWrn_Rsvd27_Q	:=	S_SPI_MNG_264.Digital_Feedback_Q	;
S_SPI_MNG_265	(Digital_Feedback_Value:=	emC_LUC[LUC_Num].SCADA.Out.GCWrn_Rsvd28	,TimeTag:=Timestamp,IV:=FALSE);	GCWrn_Rsvd28_Q	:=	S_SPI_MNG_265.Digital_Feedback_Q	;
S_SPI_MNG_266	(Digital_Feedback_Value:=	emC_LUC[LUC_Num].SCADA.Out.GCWrn_Rsvd29	,TimeTag:=Timestamp,IV:=FALSE);	GCWrn_Rsvd29_Q	:=	S_SPI_MNG_266.Digital_Feedback_Q	;
S_SPI_MNG_267	(Digital_Feedback_Value:=	emC_LUC[LUC_Num].SCADA.Out.GCWrn_Rsvd30	,TimeTag:=Timestamp,IV:=FALSE);	GCWrn_Rsvd30_Q	:=	S_SPI_MNG_267.Digital_Feedback_Q	;
S_SPI_MNG_268	(Digital_Feedback_Value:=	emC_LUC[LUC_Num].SCADA.Out.GCCriticalAlarm	,TimeTag:=Timestamp,IV:=FALSE);	GCCriticalAlarm_Q	:=	S_SPI_MNG_268.Digital_Feedback_Q	;
S_SPI_MNG_269	(Digital_Feedback_Value:=	emC_LUC[LUC_Num].SCADA.Out.GCNonCriticalAlarm	,TimeTag:=Timestamp,IV:=FALSE);	GCNonCriticalAlarm_Q	:=	S_SPI_MNG_269.Digital_Feedback_Q	;
S_SPI_MNG_270	(Digital_Feedback_Value:=	emC_LUC[LUC_Num].SCADA.Out.GCWarning	,TimeTag:=Timestamp,IV:=FALSE);	GCWarning_Q	:=	S_SPI_MNG_270.Digital_Feedback_Q	;
S_SPI_MNG_271	(Digital_Feedback_Value:=	emC_LUC[LUC_Num].SCADA.Out.GCreconnectDelay	,TimeTag:=Timestamp,IV:=FALSE);	GCreconnectDelay_Q	:=	S_SPI_MNG_271.Digital_Feedback_Q	;
S_SPI_MNG_272	(Digital_Feedback_Value:=	emC_LUC[LUC_Num].SCADA.Out.GCMomentCessation	,TimeTag:=Timestamp,IV:=FALSE);	GCMomentCessation_Q	:=	S_SPI_MNG_272.Digital_Feedback_Q	;
S_SPI_MNG_273	(Digital_Feedback_Value:=	emC_LUC[LUC_Num].SCADA.Out.GCInhibited	,TimeTag:=Timestamp,IV:=FALSE);	GCInhibited_Q	:=	S_SPI_MNG_273.Digital_Feedback_Q	;
								
								
								
								
emC_LUC[LUC_Num].SCADA.Out.PfAct	:=	emC_LUC[LUC_Num].emPs.PS.GCPF  		;
emC_LUC[LUC_Num].SCADA.Out.BatSyncUAct	:=	emC_LUC[LUC_Num].BattPLC.CtrlLo.Out.Batt_Sys.BattSysMeasure.SyncUSet  		;
emC_LUC[LUC_Num].SCADA.Out.BatSocAct	:=	emC_LUC[LUC_Num].BattPLC.CtrlLo.Out.Batt_Sys.BattSysMeasure.SocPctAct  		;
emC_LUC[LUC_Num].SCADA.Out.TempAct	:=	emC_LUC[LUC_Num].emPs.PS.TempAct  		;
emC_LUC[LUC_Num].SCADA.Out.UAct	:=	emC_LUC[LUC_Num].emPs.PS.GCUAct  		;
emC_LUC[LUC_Num].SCADA.Out.PAct	:=	emC_LUC[LUC_Num].emPs.PS.GCPAct  		;
emC_LUC[LUC_Num].SCADA.Out.QAct	:=	emC_LUC[LUC_Num].emPs.PS.GCQAct  		;
emC_LUC[LUC_Num].SCADA.Out.EAct	:=	emC_LUC[LUC_Num].emPs.PS.GCEAct  		;(*From BMS??*)
emC_LUC[LUC_Num].SCADA.Out.FAct	:=	emC_LUC[LUC_Num].emPs.PS.GCFAct  		;
(*emC_LUC[LUC_Num].SCADA.Out.GcSPNomAct	:=	emC_LUC[LUC_Num]  		;
emC_LUC[LUC_Num].SCADA.Out.GcINomAct	:=	emC_LUC[LUC_Num]  		;
emC_LUC[LUC_Num].SCADA.Out.GcUNomAct	:=	emC_LUC[LUC_Num]  		;
emC_LUC[LUC_Num].SCADA.Out.GcFNomAct	:=	emC_LUC[LUC_Num]  		;
emC_LUC[LUC_Num].SCADA.Out.GcModUNomAct	:=	emC_LUC[LUC_Num]  		;
*)
								
								
								
